C01786=1131.431,222.505,-66.418,-178.866,9.578,149.578
C01787=1131.435,222.257,-66.392,-178.868,9.575,149.578
C01788=1131.439,222.008,-66.366,-178.871,9.572,149.578
C01789=1131.445,221.760,-66.340,-178.874,9.569,149.578
C01790=1131.449,221.512,-66.313,-178.877,9.565,149.578
C01791=1131.453,221.263,-66.288,-178.880,9.562,149.578
C01792=1131.458,221.014,-66.261,-178.882,9.559,149.578
C01793=1131.462,220.765,-66.235,-178.885,9.556,149.578
C01794=1131.466,220.517,-66.209,-178.887,9.553,149.578
C01795=1131.471,220.269,-66.184,-178.890,9.550,149.578
C01796=1131.476,220.019,-66.157,-178.892,9.547,149.578
C01797=1131.480,219.771,-66.132,-178.895,9.544,149.577
C01798=1131.484,219.522,-66.105,-178.897,9.540,149.577
C01799=1131.488,219.274,-66.079,-178.899,9.537,149.577
C01800=1131.493,219.026,-66.054,-178.902,9.534,149.577
C01801=1131.498,218.776,-66.028,-178.904,9.531,149.577
C01802=1131.502,218.528,-66.002,-178.907,9.528,149.577
C01803=1131.506,218.279,-65.976,-178.910,9.525,149.577
C01804=1131.510,218.031,-65.950,-178.911,9.522,149.577
C01805=1131.515,217.783,-65.924,-178.914,9.519,149.577
C01806=1131.519,217.534,-65.899,-178.916,9.516,149.577
C01807=1131.524,217.285,-65.872,-178.918,9.513,149.576
C01808=1131.529,217.036,-65.846,-178.920,9.510,149.576
C01809=1131.533,216.788,-65.821,-178.923,9.507,149.576
C01810=1131.538,216.539,-65.795,-178.924,9.504,149.576
C01811=1131.542,216.290,-65.770,-178.927,9.501,149.576
C01812=1131.546,216.041,-65.744,-178.928,9.499,149.576
C01813=1131.551,215.793,-65.718,-178.931,9.495,149.576
C01814=1131.555,215.544,-65.693,-178.932,9.493,149.576
C01815=1131.559,215.296,-65.667,-178.934,9.490,149.575
C01816=1131.564,215.047,-65.642,-178.936,9.487,149.575
C01817=1131.569,214.798,-65.615,-178.938,9.484,149.575
C01818=1131.573,214.550,-65.589,-178.940,9.482,149.575
C01819=1131.578,214.301,-65.564,-178.942,9.479,149.575
C01820=1131.582,214.053,-65.538,-178.944,9.476,149.575
C01821=1131.587,213.804,-65.513,-178.945,9.474,149.574
C01822=1131.591,213.555,-65.487,-178.947,9.471,149.574
C01823=1131.596,213.307,-65.461,-178.949,9.469,149.574
C01824=1131.599,213.092,-65.440,-178.950,9.467,149.574
C01825=1131.603,212.878,-65.418,-178.951,9.464,149.574
C01826=1131.607,212.664,-65.395,-178.952,9.462,149.574
C01827=1131.611,212.450,-65.374,-178.954,9.460,149.574
C01828=1131.614,212.235,-65.351,-178.955,9.458,149.573
C01829=1131.618,212.021,-65.329,-178.957,9.456,149.573
C01830=1131.622,211.807,-65.307,-178.958,9.454,149.573
C01831=1131.626,211.592,-65.285,-178.960,9.452,149.573
C01832=1131.631,211.344,-65.259,-178.961,9.449,149.573
C01833=1131.634,211.096,-65.234,-178.963,9.446,149.573
C01834=1131.640,210.847,-65.210,-178.965,9.444,149.573
C01835=1131.644,210.598,-65.184,-178.967,9.442,149.573
C01836=1131.648,210.349,-65.158,-178.969,9.439,149.573
C01837=1131.653,210.101,-65.133,-178.970,9.437,149.572
C01838=1131.657,209.852,-65.107,-178.972,9.434,149.572
C01839=1131.662,209.603,-65.082,-178.975,9.431,149.572
C01840=1131.666,209.355,-65.057,-178.976,9.429,149.572
C01841=1131.671,209.106,-65.031,-178.979,9.427,149.572
C01842=1131.675,208.857,-65.005,-178.981,9.424,149.572
C01843=1131.680,208.608,-64.980,-178.983,9.422,149.572
C01844=1131.684,208.360,-64.955,-178.985,9.419,149.572
C01845=1131.689,208.112,-64.929,-178.988,9.416,149.572
C01846=1131.694,207.862,-64.904,-178.990,9.414,149.572
C01847=1131.697,207.614,-64.879,-178.992,9.411,149.572
C01848=1131.702,207.366,-64.854,-178.995,9.408,149.572
C01849=1131.706,207.116,-64.829,-178.997,9.406,149.572
C01850=1131.711,206.868,-64.803,-179.000,9.403,149.572
C01851=1131.715,206.619,-64.778,-179.003,9.400,149.572
C01852=1131.721,206.371,-64.753,-179.005,9.397,149.572
C01853=1131.725,206.122,-64.727,-179.008,9.395,149.573
C01854=1131.729,205.874,-64.702,-179.011,9.392,149.573
C01855=1131.733,205.624,-64.677,-179.013,9.389,149.573
C01856=1131.738,205.376,-64.652,-179.016,9.387,149.573
C01857=1131.743,205.127,-64.627,-179.019,9.384,149.573
C01858=1131.747,204.878,-64.601,-179.022,9.381,149.573
C01859=1131.751,204.630,-64.577,-179.024,9.378,149.573
C01860=1131.756,204.381,-64.551,-179.027,9.375,149.573
C01861=1131.761,204.132,-64.527,-179.031,9.372,149.573
C01862=1131.765,203.883,-64.501,-179.034,9.369,149.573
C01863=1131.770,203.635,-64.476,-179.036,9.366,149.573
C01864=1131.774,203.386,-64.451,-179.039,9.363,149.574
C01865=1131.779,203.137,-64.426,-179.043,9.360,149.574
C01866=1131.783,202.889,-64.401,-179.046,9.357,149.574
C01867=1131.787,202.640,-64.377,-179.050,9.353,149.574
C01868=1131.792,202.391,-64.351,-179.053,9.351,149.574
C01869=1131.797,202.143,-64.326,-179.056,9.347,149.574
C01870=1131.801,201.894,-64.302,-179.059,9.344,149.574
C01871=1131.805,201.646,-64.276,-179.063,9.341,149.575
C01872=1131.810,201.397,-64.252,-179.066,9.337,149.575
C01873=1131.814,201.148,-64.227,-179.070,9.334,149.575
C01874=1131.819,200.900,-64.202,-179.073,9.331,149.575
C01875=1131.823,200.650,-64.177,-179.077,9.328,149.575
C01876=1131.828,200.402,-64.153,-179.080,9.324,149.575
C01877=1131.833,200.152,-64.128,-179.084,9.321,149.576
C01878=1131.837,199.905,-64.103,-179.088,9.317,149.576
C01879=1131.842,199.656,-64.078,-179.091,9.314,149.576
C01880=1131.845,199.440,-64.057,-179.095,9.310,149.576
C01881=1131.849,199.227,-64.036,-179.098,9.308,149.576
C01882=1131.853,199.012,-64.015,-179.101,9.304,149.576
C01883=1131.857,198.798,-63.993,-179.104,9.301,149.576
C01884=1131.861,198.583,-63.972,-179.108,9.298,149.577
C01885=1131.864,198.369,-63.950,-179.111,9.295,149.577
C01886=1131.868,198.155,-63.930,-179.114,9.292,149.577
C01887=1131.872,197.941,-63.908,-179.118,9.288,149.577
C01888=1131.877,197.692,-63.884,-179.122,9.285,149.577
C01889=1131.882,197.443,-63.860,-179.126,9.281,149.578
C01890=1131.886,197.194,-63.834,-179.130,9.277,149.578
C01891=1131.890,196.946,-63.810,-179.134,9.273,149.578
C01892=1131.896,196.697,-63.786,-179.138,9.269,149.578
C01893=1131.899,196.448,-63.761,-179.142,9.265,149.578
C01894=1131.904,196.199,-63.737,-179.146,9.261,149.578
C01895=1131.909,195.951,-63.713,-179.147,9.259,149.578
C01896=1131.913,195.702,-63.688,-179.148,9.256,149.578
C01897=1131.918,195.453,-63.663,-179.150,9.254,149.578
C01898=1131.923,195.204,-63.640,-179.152,9.251,149.577
C01899=1131.927,194.955,-63.616,-179.153,9.248,149.577
C01900=1131.931,194.706,-63.591,-179.155,9.246,149.577
C01901=1131.936,194.458,-63.567,-179.156,9.244,149.577
C01902=1131.940,194.209,-63.543,-179.157,9.241,149.577
C01903=1131.945,193.960,-63.518,-179.159,9.239,149.577
C01904=1131.949,193.711,-63.494,-179.161,9.236,149.576
C01905=1131.954,193.463,-63.470,-179.163,9.234,149.576
C01906=1131.959,193.213,-63.446,-179.164,9.231,149.576
C01907=1131.963,192.965,-63.422,-179.166,9.229,149.576
C01908=1131.967,192.716,-63.397,-179.167,9.226,149.576
C01909=1131.972,192.467,-63.372,-179.169,9.224,149.576
C01910=1131.977,192.219,-63.348,-179.171,9.221,149.576
C01911=1131.981,191.970,-63.324,-179.173,9.218,149.576
C01912=1131.986,191.720,-63.300,-179.175,9.216,149.576
C01913=1131.990,191.472,-63.276,-179.177,9.213,149.575
C01914=1131.995,191.224,-63.252,-179.179,9.211,149.575
C01915=1131.999,190.975,-63.228,-179.181,9.208,149.575
C01916=1132.005,190.726,-63.204,-179.183,9.205,149.575
C01917=1132.008,190.477,-63.179,-179.184,9.203,149.575
C01918=1132.013,190.228,-63.155,-179.187,9.200,149.575
C01919=1132.018,189.980,-63.131,-179.189,9.197,149.575
C01920=1132.023,189.731,-63.107,-179.191,9.195,149.575
C01921=1132.027,189.482,-63.083,-179.193,9.192,149.575
C01922=1132.031,189.234,-63.059,-179.195,9.189,149.575
C01923=1132.035,188.984,-63.035,-179.198,9.186,149.575
C01924=1132.041,188.735,-63.011,-179.200,9.184,149.575
C01925=1132.045,188.487,-62.987,-179.202,9.181,149.575
C01926=1132.050,188.238,-62.963,-179.205,9.178,149.575
C01927=1132.054,187.989,-62.939,-179.207,9.176,149.575
C01928=1132.058,187.741,-62.915,-179.209,9.172,149.575
C01929=1132.063,187.491,-62.891,-179.212,9.169,149.575
C01930=1132.068,187.243,-62.867,-179.213,9.167,149.574
C01931=1132.072,186.993,-62.843,-179.216,9.164,149.574
C01932=1132.077,186.745,-62.819,-179.219,9.161,149.574
C01933=1132.081,186.496,-62.796,-179.221,9.158,149.574
C01934=1132.086,186.248,-62.772,-179.224,9.155,149.574
C01935=1132.090,185.999,-62.748,-179.226,9.153,149.574
C01936=1132.095,185.784,-62.728,-179.228,9.149,149.574
C01937=1132.098,185.569,-62.707,-179.230,9.147,149.574
C01938=1132.102,185.355,-62.686,-179.233,9.144,149.574
C01939=1132.106,185.140,-62.666,-179.235,9.142,149.574
C01940=1132.111,184.926,-62.645,-179.237,9.140,149.574
C01941=1132.114,184.712,-62.625,-179.240,9.137,149.574
C01942=1132.118,184.498,-62.604,-179.241,9.134,149.574
C01943=1132.122,184.282,-62.584,-179.244,9.131,149.574
C01944=1132.126,184.034,-62.560,-179.247,9.128,149.574
C01945=1132.131,183.785,-62.537,-179.249,9.125,149.575
C01946=1132.136,183.536,-62.513,-179.253,9.121,149.574
C01947=1132.140,183.287,-62.489,-179.255,9.118,149.574
C01948=1132.145,183.038,-62.466,-179.258,9.116,149.575
C01949=1132.149,182.790,-62.442,-179.261,9.113,149.575
C01950=1132.154,182.541,-62.418,-179.264,9.109,149.574
C01951=1132.159,182.292,-62.395,-179.267,9.106,149.575
C01952=1132.163,182.043,-62.371,-179.269,9.103,149.575
C01953=1132.168,181.794,-62.348,-179.272,9.099,149.575
C01954=1132.173,181.545,-62.324,-179.275,9.096,149.575
C01955=1132.177,181.297,-62.300,-179.279,9.092,149.575
C01956=1132.182,181.048,-62.277,-179.282,9.090,149.575
C01957=1132.186,180.799,-62.254,-179.285,9.086,149.575
C01958=1132.191,180.550,-62.230,-179.288,9.082,149.575
C01959=1132.195,180.302,-62.206,-179.291,9.079,149.575
C01960=1132.199,180.053,-62.183,-179.294,9.075,149.575
C01961=1132.204,179.804,-62.160,-179.298,9.072,149.575
C01962=1132.209,179.555,-62.137,-179.300,9.069,149.575
C01963=1132.214,179.306,-62.113,-179.304,9.065,149.575
C01964=1132.218,179.057,-62.090,-179.306,9.062,149.575
C01965=1132.223,178.808,-62.067,-179.308,9.058,149.575
C01966=1132.227,178.559,-62.042,-179.311,9.055,149.575
C01967=1132.231,178.310,-62.020,-179.312,9.053,149.575
C01968=1132.236,178.061,-61.996,-179.315,9.050,149.575
C01969=1132.241,177.812,-61.973,-179.317,9.047,149.575
C01970=1132.245,177.563,-61.950,-179.319,9.044,149.574
C01971=1132.250,177.314,-61.926,-179.321,9.041,149.574
C01972=1132.254,177.066,-61.903,-179.323,9.038,149.574
C01973=1132.259,176.817,-61.880,-179.325,9.035,149.574
C01974=1132.264,176.568,-61.857,-179.327,9.033,149.574
C01975=1132.269,176.319,-61.834,-179.330,9.029,149.574
C01976=1132.273,176.071,-61.811,-179.332,9.026,149.574
C01977=1132.277,175.821,-61.788,-179.334,9.024,149.574
C01978=1132.282,175.572,-61.764,-179.336,9.020,149.574
C01979=1132.287,175.323,-61.741,-179.338,9.017,149.573
C01980=1132.291,175.075,-61.718,-179.340,9.015,149.573
C01981=1132.296,174.826,-61.695,-179.343,9.012,149.573
C01982=1132.301,174.577,-61.672,-179.345,9.008,149.573
C01983=1132.305,174.328,-61.648,-179.347,9.005,149.573
C01984=1132.310,174.079,-61.626,-179.349,9.003,149.573
C01985=1132.314,173.830,-61.603,-179.352,9.000,149.573
C01986=1132.319,173.581,-61.580,-179.354,8.996,149.573
C01987=1132.323,173.332,-61.557,-179.356,8.994,149.573
C01988=1132.328,173.084,-61.534,-179.358,8.991,149.573
C01989=1132.333,172.835,-61.511,-179.361,8.988,149.573
C01990=1132.337,172.586,-61.488,-179.363,8.984,149.572
C01991=1132.342,172.336,-61.465,-179.365,8.981,149.572
C01992=1132.346,172.123,-61.445,-179.367,8.979,149.572
C01993=1132.350,171.908,-61.425,-179.369,8.976,149.572
C01994=1132.354,171.693,-61.406,-179.371,8.974,149.572
C01995=1132.358,171.478,-61.386,-179.373,8.970,149.572
C01996=1132.362,171.264,-61.366,-179.375,8.968,149.572
C01997=1132.366,171.049,-61.346,-179.377,8.966,149.572
C01998=1132.370,170.835,-61.327,-179.380,8.963,149.572
C01999=1132.373,170.620,-61.307,-179.381,8.960,149.572
C02000=1132.379,170.371,-61.284,-179.383,8.957,149.572
C02001=1132.383,170.122,-61.261,-179.386,8.954,149.572
C02002=1132.388,169.873,-61.239,-179.388,8.951,149.572
C02003=1132.392,169.624,-61.216,-179.390,8.948,149.572
C02004=1132.397,169.376,-61.193,-179.393,8.945,149.571
C02005=1132.402,169.126,-61.171,-179.395,8.942,149.571
C02006=1132.406,168.878,-61.148,-179.398,8.939,149.571
C02007=1132.411,168.629,-61.125,-179.400,8.936,149.571
C02008=1132.415,168.380,-61.103,-179.402,8.932,149.571
C02009=1132.420,168.131,-61.079,-179.405,8.929,149.571
C02010=1132.424,167.882,-61.057,-179.407,8.926,149.571
C02011=1132.430,167.633,-61.034,-179.410,8.923,149.571
C02012=1132.434,167.384,-61.012,-179.412,8.920,149.571
C02013=1132.439,167.135,-60.989,-179.414,8.916,149.571
C02014=1132.443,166.887,-60.967,-179.417,8.913,149.571
C02015=1132.448,166.637,-60.944,-179.419,8.910,149.571
C02016=1132.452,166.388,-60.921,-179.422,8.907,149.571
C02017=1132.458,166.139,-60.899,-179.424,8.903,149.570
C02018=1132.462,165.891,-60.876,-179.427,8.900,149.570
C02019=1132.466,165.641,-60.854,-179.429,8.897,149.570
C02020=1132.471,165.393,-60.831,-179.432,8.894,149.570
C02021=1132.476,165.144,-60.809,-179.434,8.891,149.570
C02022=1132.481,164.894,-60.786,-179.436,8.887,149.570
C02023=1132.485,164.646,-60.764,-179.439,8.884,149.570
C02024=1132.489,164.397,-60.742,-179.441,8.881,149.570
C02025=1132.494,164.148,-60.719,-179.444,8.878,149.570
C02026=1132.499,163.899,-60.697,-179.446,8.875,149.570
C02027=1132.503,163.650,-60.675,-179.448,8.872,149.570
C02028=1132.508,163.401,-60.652,-179.451,8.868,149.570
C02029=1132.513,163.152,-60.630,-179.453,8.865,149.570
C02030=1132.517,162.903,-60.607,-179.457,8.861,149.569
C02031=1132.522,162.654,-60.585,-179.459,8.858,149.569
C02032=1132.527,162.405,-60.563,-179.461,8.855,149.569
C02033=1132.531,162.156,-60.541,-179.464,8.852,149.569
C02034=1132.536,161.907,-60.518,-179.466,8.849,149.569
C02035=1132.540,161.658,-60.496,-179.468,8.845,149.569
C02036=1132.545,161.409,-60.474,-179.472,8.841,149.569
C02037=1132.550,161.160,-60.452,-179.474,8.838,149.569
C02038=1132.555,160.912,-60.429,-179.477,8.835,149.569
C02039=1132.559,160.662,-60.407,-179.479,8.832,149.569
C02040=1132.563,160.413,-60.385,-179.482,8.828,149.569
C02041=1132.568,160.164,-60.363,-179.484,8.825,149.569
C02042=1132.573,159.915,-60.341,-179.487,8.821,149.568
C02043=1132.578,159.667,-60.318,-179.489,8.818,149.568
C02044=1132.582,159.417,-60.296,-179.492,8.814,149.568
C02045=1132.587,159.169,-60.274,-179.495,8.811,149.568
C02046=1132.591,158.919,-60.252,-179.497,8.808,149.568
C02047=1132.596,158.671,-60.231,-179.500,8.804,149.568
C02048=1132.604,158.252,-60.193,-179.504,8.798,149.568
C02049=1132.612,157.833,-60.156,-179.508,8.792,149.568
C02050=1132.620,157.416,-60.119,-179.513,8.786,149.568
C02051=1132.628,156.997,-60.082,-179.517,8.780,149.567
C02052=1132.632,156.748,-60.061,-179.520,8.777,149.567
C02053=1132.637,156.499,-60.039,-179.523,8.773,149.567
C02054=1132.642,156.250,-60.017,-179.525,8.770,149.567
C02055=1132.646,156.001,-59.995,-179.528,8.766,149.567
C02056=1132.651,155.752,-59.973,-179.531,8.763,149.567
C02057=1132.655,155.503,-59.951,-179.534,8.759,149.567
C02058=1132.660,155.254,-59.930,-179.536,8.755,149.567
C02059=1132.665,155.006,-59.908,-179.538,8.752,149.567
C02060=1132.669,154.756,-59.887,-179.542,8.748,149.567
C02061=1132.674,154.507,-59.865,-179.544,8.744,149.566
C02062=1132.678,154.258,-59.843,-179.547,8.741,149.566
C02063=1132.683,154.009,-59.821,-179.550,8.737,149.566
C02064=1132.688,153.760,-59.799,-179.552,8.734,149.566
C02065=1132.692,153.511,-59.777,-179.555,8.730,149.566
C02066=1132.698,153.262,-59.756,-179.557,8.726,149.566
C02067=1132.703,153.013,-59.735,-179.560,8.722,149.566
C02068=1132.707,152.764,-59.713,-179.563,8.719,149.566
C02069=1132.712,152.515,-59.691,-179.566,8.715,149.566
C02070=1132.717,152.266,-59.670,-179.569,8.711,149.566
C02071=1132.721,152.016,-59.648,-179.571,8.708,149.565
C02072=1132.726,151.768,-59.626,-179.574,8.704,149.565
C02073=1132.731,151.519,-59.605,-179.577,8.700,149.565
C02074=1132.735,151.269,-59.583,-179.579,8.696,149.565
C02075=1132.740,151.021,-59.562,-179.582,8.693,149.565
C02076=1132.745,150.772,-59.541,-179.585,8.688,149.565
C02077=1132.749,150.522,-59.519,-179.588,8.685,149.565
C02078=1132.754,150.274,-59.497,-179.590,8.681,149.565
C02079=1132.759,150.024,-59.477,-179.594,8.677,149.564
C02080=1132.782,148.793,-59.374,-178.796,7.149,148.985
C02081=1132.787,148.545,-59.352,-178.799,7.147,148.985
C02082=1132.792,148.296,-59.332,-178.802,7.145,148.985
C02083=1132.796,148.046,-59.310,-178.805,7.143,148.986
C02084=1132.801,147.797,-59.289,-178.807,7.141,148.986
C02085=1132.805,147.548,-59.268,-178.811,7.139,148.986
C02086=1132.811,147.299,-59.247,-178.813,7.137,148.987
C02087=1132.816,147.050,-59.226,-178.816,7.135,148.987
C02088=1132.820,146.801,-59.205,-178.819,7.132,148.987
C02089=1132.825,146.552,-59.184,-178.822,7.131,148.988
C02090=1132.830,146.303,-59.164,-178.824,7.129,148.988
C02091=1132.834,146.053,-59.143,-178.828,7.127,148.988
C02092=1132.839,145.805,-59.121,-178.830,7.125,148.989
C02093=1132.843,145.556,-59.100,-178.833,7.123,148.989
C02094=1132.849,145.306,-59.080,-178.836,7.120,148.989
C02095=1132.853,145.057,-59.059,-178.839,7.119,148.990
C02096=1132.858,144.808,-59.038,-178.841,7.117,148.990
C02097=1132.863,144.559,-59.018,-178.845,7.114,148.991
C02098=1132.867,144.311,-58.996,-178.847,7.113,148.991
C02099=1132.872,144.062,-58.976,-178.850,7.111,148.991
C02100=1132.877,143.812,-58.955,-178.853,7.108,148.991
C02101=1132.882,143.563,-58.934,-178.856,7.106,148.992
C02102=1132.886,143.313,-58.913,-178.858,7.105,148.992
C02103=1132.891,143.065,-58.893,-178.862,7.102,148.993
C02104=1132.896,142.815,-58.872,-178.864,7.101,148.993
C02105=1132.900,142.566,-58.851,-178.867,7.098,148.993
C02106=1132.905,142.317,-58.830,-178.869,7.097,148.994
C02107=1132.910,142.068,-58.810,-178.873,7.094,148.994
C02108=1132.915,141.819,-58.789,-178.875,7.093,148.994
C02109=1132.919,141.570,-58.769,-178.878,7.091,148.995
C02110=1132.924,141.321,-58.748,-178.881,7.088,148.995
C02111=1132.929,141.072,-58.727,-178.884,7.087,148.995
C02112=1132.933,140.823,-58.707,-178.886,7.085,148.996
C02113=1132.939,140.573,-58.686,-178.889,7.083,148.996
C02114=1132.943,140.325,-58.666,-178.892,7.080,148.996
C02115=1132.947,140.076,-58.645,-178.895,7.079,148.997
C02116=1132.953,139.826,-58.624,-178.898,7.077,148.997
C02117=1132.957,139.577,-58.604,-178.901,7.075,148.998
C02118=1132.962,139.328,-58.584,-178.904,7.073,148.998
C02119=1132.967,139.079,-58.563,-178.907,7.071,148.998
C02120=1132.971,138.830,-58.543,-178.909,7.069,148.999
C02121=1132.976,138.581,-58.523,-178.912,7.067,148.999
C02122=1132.981,138.331,-58.502,-178.915,7.065,148.999
C02123=1132.985,138.082,-58.481,-178.918,7.063,149.000
C02124=1132.990,137.833,-58.461,-178.920,7.062,149.000
C02125=1132.995,137.584,-58.440,-178.924,7.059,149.000
C02126=1133.000,137.335,-58.420,-178.926,7.057,149.001
C02127=1133.004,137.086,-58.400,-178.929,7.056,149.001
C02128=1133.010,136.837,-58.379,-178.931,7.054,149.001
C02129=1133.014,136.588,-58.359,-178.935,7.051,149.002
C02130=1133.019,136.339,-58.339,-178.937,7.049,149.002
C02131=1133.024,136.090,-58.319,-178.940,7.048,149.003
C02132=1133.029,135.840,-58.298,-178.943,7.046,149.003
C02133=1133.033,135.591,-58.278,-178.946,7.044,149.003
C02134=1133.038,135.342,-58.258,-178.949,7.042,149.004
C02135=1133.042,135.093,-58.237,-178.952,7.040,149.004
C02136=1133.048,134.844,-58.217,-178.954,7.038,149.005
C02137=1133.052,134.594,-58.197,-178.958,7.036,149.005
C02138=1133.057,134.346,-58.177,-178.960,7.034,149.005
C02139=1133.062,134.097,-58.156,-178.963,7.032,149.005
C02140=1133.067,133.847,-58.137,-178.965,7.031,149.006
C02141=1133.072,133.598,-58.116,-178.969,7.028,149.006
C02142=1133.076,133.349,-58.096,-178.971,7.026,149.007
C02143=1133.081,133.100,-58.076,-178.974,7.025,149.007
C02144=1133.085,132.851,-58.055,-178.977,7.023,149.007
C02145=1133.091,132.602,-58.036,-178.980,7.021,149.008
C02146=1133.095,132.353,-58.016,-178.983,7.019,149.008
C02147=1133.100,132.103,-57.996,-178.986,7.017,149.009
C02148=1133.105,131.854,-57.975,-178.988,7.015,149.009
C02149=1133.110,131.585,-57.954,-178.991,7.014,149.009
C02150=1133.115,131.317,-57.932,-178.994,7.011,149.010
C02151=1133.120,131.048,-57.911,-178.997,7.010,149.010
C02152=1133.125,130.780,-57.890,-179.000,7.007,149.011
C02153=1133.130,130.531,-57.869,-179.003,7.005,149.011
C02154=1133.136,130.282,-57.849,-179.006,7.004,149.011
C02155=1133.140,130.033,-57.829,-179.009,7.002,149.012
C02156=1133.145,129.783,-57.809,-179.012,6.999,149.012
C02157=1133.149,129.534,-57.789,-179.014,6.997,149.012
C02158=1133.155,129.285,-57.770,-179.017,6.996,149.013
C02159=1133.159,129.036,-57.750,-179.020,6.994,149.013
C02160=1133.164,128.787,-57.730,-179.022,6.992,149.014
C02161=1133.169,128.537,-57.710,-179.026,6.990,149.014
C02162=1133.174,128.289,-57.690,-179.028,6.988,149.014
C02163=1133.178,128.039,-57.670,-179.031,6.987,149.015
C02164=1133.183,127.790,-57.651,-179.034,6.985,149.015
C02165=1133.188,127.541,-57.630,-179.037,6.983,149.016
C02166=1133.193,127.292,-57.611,-179.039,6.981,149.016
C02167=1133.198,127.042,-57.591,-179.043,6.979,149.016
C02168=1133.202,126.793,-57.571,-179.045,6.977,149.017
C02169=1133.207,126.544,-57.551,-179.048,6.976,149.017
C02170=1133.212,126.295,-57.532,-179.051,6.974,149.018
C02171=1133.217,126.045,-57.512,-179.054,6.972,149.018
C02172=1133.221,125.796,-57.492,-179.056,6.971,149.018
C02173=1133.226,125.548,-57.473,-179.060,6.968,149.019
C02174=1133.231,125.298,-57.454,-179.062,6.966,149.019
C02175=1133.235,125.049,-57.434,-179.065,6.965,149.019
C02176=1133.240,124.800,-57.414,-179.068,6.963,149.020
C02177=1133.245,124.551,-57.394,-179.071,6.961,149.020
C02178=1133.250,124.301,-57.375,-179.073,6.960,149.021
C02179=1133.255,124.052,-57.355,-179.076,6.957,149.021
C02180=1133.260,123.803,-57.336,-179.079,6.955,149.021
C02181=1133.264,123.554,-57.315,-179.082,6.953,149.022
C02182=1133.268,123.305,-57.296,-179.084,6.952,149.022
C02183=1133.274,123.056,-57.277,-179.087,6.950,149.022
C02184=1133.279,122.806,-57.257,-179.090,6.948,149.023
C02185=1133.283,122.557,-57.238,-179.092,6.947,149.023
C02186=1133.289,122.308,-57.218,-179.096,6.944,149.024
C02187=1133.293,122.058,-57.199,-179.099,6.943,149.024
C02188=1133.298,121.810,-57.180,-179.101,6.941,149.024
C02189=1133.303,121.560,-57.160,-179.104,6.939,149.025
C02190=1133.307,121.311,-57.140,-179.107,6.937,149.025
C02191=1133.313,121.062,-57.121,-179.109,6.936,149.026
C02192=1133.317,120.813,-57.101,-179.112,6.934,149.026
C02193=1133.322,120.564,-57.082,-179.115,6.932,149.026
C02194=1133.327,120.315,-57.063,-179.118,6.930,149.027
C02195=1133.331,120.065,-57.043,-179.121,6.928,149.027
C02196=1133.337,119.816,-57.024,-179.124,6.927,149.028
C02197=1133.341,119.567,-57.005,-179.126,6.925,149.028
C02198=1133.346,119.318,-56.985,-179.129,6.923,149.029
C02199=1133.351,119.069,-56.966,-179.132,6.922,149.029
C02200=1133.356,118.819,-56.948,-179.135,6.920,149.029
C02201=1133.360,118.570,-56.928,-179.137,6.918,149.030
C02202=1133.365,118.320,-56.908,-179.140,6.916,149.030
C02203=1133.371,118.071,-56.889,-179.143,6.914,149.031
C02204=1133.375,117.822,-56.870,-179.146,6.912,149.031
C02205=1133.380,117.573,-56.851,-179.149,6.911,149.031
C02206=1133.385,117.324,-56.831,-179.152,6.909,149.032
C02207=1133.389,117.075,-56.812,-179.154,6.907,149.032
C02208=1133.394,116.826,-56.793,-179.157,6.906,149.033
C02209=1133.400,116.576,-56.774,-179.160,6.904,149.033
C02210=1133.404,116.327,-56.755,-179.163,6.902,149.033
C02211=1133.409,116.078,-56.736,-179.165,6.901,149.034
C02212=1133.413,115.829,-56.717,-179.168,6.899,149.034
C02213=1133.418,115.580,-56.697,-179.171,6.897,149.035
C02214=1133.423,115.330,-56.679,-179.174,6.895,149.035
C02215=1133.428,115.081,-56.660,-179.177,6.893,149.035
C02216=1133.433,114.832,-56.640,-179.180,6.891,149.036
C02217=1133.438,114.583,-56.621,-179.183,6.890,149.036
C02218=1133.442,114.333,-56.603,-179.185,6.888,149.037
C02219=1133.448,114.084,-56.583,-179.188,6.887,149.037
C02220=1133.452,113.835,-56.564,-179.191,6.885,149.038
C02221=1133.457,113.586,-56.545,-179.194,6.883,149.038
C02222=1133.462,113.337,-56.527,-179.196,6.882,149.038
C02223=1133.467,113.087,-56.507,-179.199,6.880,149.039
C02224=1133.471,112.838,-56.489,-179.202,6.878,149.039
C02225=1133.476,112.588,-56.470,-179.205,6.877,149.040
C02226=1133.482,112.339,-56.450,-179.207,6.875,149.040
C02227=1133.486,112.090,-56.431,-179.210,6.873,149.040
C02228=1133.491,111.841,-56.413,-179.213,6.872,149.041
C02229=1133.496,111.592,-56.394,-179.216,6.870,149.041
C02230=1133.501,111.342,-56.375,-179.219,6.867,149.042
C02231=1133.506,111.093,-56.356,-179.222,6.866,149.042
C02232=1133.510,110.844,-56.337,-179.224,6.864,149.043
C02233=1133.515,110.595,-56.319,-179.227,6.862,149.043
C02234=1133.520,110.346,-56.300,-179.230,6.861,149.043
C02235=1133.525,110.096,-56.281,-179.233,6.859,149.044
C02236=1133.530,109.847,-56.262,-179.235,6.857,149.044
C02237=1133.535,109.597,-56.243,-179.238,6.856,149.045
C02238=1133.539,109.349,-56.225,-179.241,6.854,149.045
C02239=1133.545,109.099,-56.206,-179.243,6.852,149.045
C02240=1133.549,108.850,-56.187,-179.247,6.851,149.046
C02241=1133.554,108.601,-56.169,-179.249,6.849,149.046
C02242=1133.559,108.352,-56.150,-179.252,6.848,149.047
C02243=1133.563,108.102,-56.132,-179.255,6.846,149.047
C02244=1133.569,107.853,-56.112,-179.258,6.844,149.048
C02245=1133.574,107.604,-56.094,-179.260,6.843,149.048
C02246=1133.578,107.355,-56.075,-179.263,6.841,149.048
C02247=1133.583,107.105,-56.057,-179.266,6.839,149.049
C02248=1133.588,106.856,-56.039,-179.269,6.838,149.049
C02249=1133.592,106.607,-56.020,-179.271,6.836,149.050
C02250=1133.598,106.357,-56.001,-179.274,6.834,149.050
C02251=1133.603,106.108,-55.983,-179.277,6.833,149.051
C02252=1133.607,105.859,-55.964,-179.279,6.831,149.051
C02253=1133.613,105.590,-55.944,-179.283,6.830,149.052
C02254=1133.618,105.322,-55.925,-179.286,6.827,149.052
C02255=1133.623,105.054,-55.904,-179.289,6.826,149.052
C02256=1133.628,104.786,-55.884,-179.292,6.824,149.053
C02257=1133.633,104.536,-55.866,-179.294,6.822,149.053
C02258=1133.638,104.286,-55.847,-179.297,6.821,149.054
C02259=1133.643,104.038,-55.829,-179.300,6.819,149.054
C02260=1133.647,103.788,-55.810,-179.303,6.818,149.055
C02261=1133.652,103.539,-55.792,-179.306,6.816,149.055
C02262=1133.658,103.289,-55.774,-179.308,6.814,149.056
C02263=1133.662,103.041,-55.755,-179.311,6.813,149.056
C02264=1133.667,102.791,-55.737,-179.314,6.811,149.056
C02265=1133.672,102.542,-55.719,-179.317,6.809,149.057
C02266=1133.677,102.292,-55.700,-179.319,6.808,149.057
C02267=1133.682,102.044,-55.682,-179.322,6.806,149.058
C02268=1133.687,101.794,-55.664,-179.325,6.804,149.058
C02269=1133.691,101.545,-55.645,-179.328,6.803,149.059
C02270=1133.696,101.295,-55.627,-179.331,6.801,149.059
C02271=1133.702,101.046,-55.609,-179.334,6.800,149.059
C02272=1133.707,100.797,-55.591,-179.336,6.798,149.060
C02273=1133.711,100.548,-55.573,-179.339,6.796,149.060
C02274=1133.715,100.298,-55.554,-179.342,6.795,149.061
C02275=1133.720,100.049,-55.536,-179.344,6.793,149.061
C02276=1133.725,99.800,-55.518,-179.347,6.792,149.062
C02277=1133.730,99.551,-55.500,-179.349,6.790,149.062
C02278=1133.736,99.301,-55.481,-179.352,6.789,149.062
C02279=1133.740,99.051,-55.463,-179.355,6.787,149.063
C02280=1133.745,98.802,-55.445,-179.358,6.786,149.063
C02281=1133.750,98.553,-55.427,-179.361,6.784,149.064
C02282=1133.755,98.304,-55.409,-179.364,6.782,149.064
C02283=1133.760,98.055,-55.391,-179.366,6.781,149.065
C02284=1133.765,97.806,-55.373,-179.369,6.779,149.065
C02285=1133.770,97.556,-55.355,-179.372,6.777,149.066
C02286=1133.774,97.307,-55.337,-179.374,6.776,149.066
C02287=1133.779,97.057,-55.319,-179.377,6.774,149.066
C02288=1133.784,96.808,-55.301,-179.380,6.773,149.067
C02289=1133.789,96.559,-55.283,-179.383,6.771,149.067
C02290=1133.794,96.310,-55.265,-179.386,6.769,149.068
C02291=1133.799,96.061,-55.247,-179.389,6.768,149.068
C02292=1133.803,95.811,-55.229,-179.391,6.766,149.069
C02293=1133.808,95.562,-55.211,-179.394,6.765,149.069
C02294=1133.813,95.313,-55.193,-179.396,6.764,149.070
C02295=1133.818,95.063,-55.175,-179.400,6.762,149.070
C02296=1133.823,94.813,-55.157,-179.402,6.761,149.071
C02297=1133.828,94.564,-55.139,-179.405,6.759,149.071
C02298=1133.833,94.315,-55.121,-179.408,6.757,149.071
C02299=1133.838,94.066,-55.103,-179.410,6.756,149.072
C02300=1133.842,93.817,-55.085,-179.413,6.754,149.072
C02301=1133.848,93.567,-55.068,-179.416,6.752,149.073
C02302=1133.853,93.318,-55.050,-179.419,6.751,149.073
C02303=1133.857,93.069,-55.032,-179.422,6.749,149.074
C02304=1133.862,92.819,-55.014,-179.424,6.748,149.074
C02305=1133.867,92.570,-54.996,-179.427,6.747,149.075
C02306=1133.873,92.320,-54.979,-179.430,6.745,149.075
C02307=1133.877,92.071,-54.961,-179.432,6.744,149.075
C02308=1133.882,91.822,-54.943,-179.435,6.742,149.076
C02309=1133.887,91.573,-54.925,-179.438,6.740,149.076
C02310=1133.892,91.323,-54.908,-179.441,6.739,149.077
C02311=1133.897,91.074,-54.890,-179.444,6.737,149.077
C02312=1133.902,90.825,-54.872,-179.446,6.736,149.078
C02313=1133.906,90.576,-54.854,-179.449,6.735,149.078
C02314=1133.912,90.326,-54.837,-179.451,6.733,149.079
C02315=1133.917,90.077,-54.819,-179.454,6.731,149.079
C02316=1133.922,89.828,-54.801,-179.457,6.730,149.080
C02317=1133.926,89.578,-54.784,-179.460,6.728,149.080
C02318=1133.931,89.329,-54.766,-179.463,6.727,149.081
C02319=1133.936,89.079,-54.749,-179.466,6.725,149.081
C02320=1133.941,88.830,-54.731,-179.468,6.723,149.081
C02321=1133.946,88.581,-54.713,-179.470,6.723,149.082
C02322=1133.951,88.331,-54.696,-179.473,6.721,149.082
C02323=1133.955,88.082,-54.678,-179.476,6.720,149.083
C02324=1133.961,87.832,-54.661,-179.479,6.718,149.083
C02325=1133.965,87.583,-54.643,-179.482,6.716,149.084
C02326=1133.970,87.334,-54.625,-179.485,6.715,149.084
C02327=1133.975,87.085,-54.609,-179.487,6.713,149.085
C02328=1133.980,86.835,-54.591,-179.490,6.711,149.085
C02329=1133.985,86.586,-54.573,-179.493,6.711,149.086
C02330=1133.990,86.337,-54.555,-179.496,6.709,149.086
C02331=1133.994,86.087,-54.539,-179.498,6.708,149.087
C02332=1133.999,85.838,-54.521,-179.501,6.706,149.087
C02333=1134.005,85.589,-54.504,-179.504,6.704,149.087
C02334=1134.010,85.340,-54.486,-179.506,6.703,149.088
C02335=1134.015,85.090,-54.469,-179.509,6.702,149.088
C02336=1134.019,84.841,-54.451,-179.512,6.700,149.089
C02337=1134.025,84.591,-54.434,-179.515,6.699,149.089
C02338=1134.029,84.342,-54.417,-179.517,6.697,149.090
C02339=1134.034,84.092,-54.399,-179.520,6.695,149.090
C02340=1134.039,83.843,-54.382,-179.523,6.694,149.091
C02341=1134.043,83.594,-54.365,-179.525,6.693,149.091
C02342=1134.049,83.345,-54.348,-179.528,6.692,149.092
C02343=1134.054,83.095,-54.330,-179.531,6.690,149.092
C02344=1134.059,82.846,-54.313,-179.534,6.688,149.092
C02345=1134.064,82.596,-54.296,-179.536,6.687,149.093
C02346=1134.068,82.347,-54.279,-179.540,6.685,149.094
C02347=1134.073,82.098,-54.261,-179.542,6.685,149.094
C02348=1134.078,81.848,-54.244,-179.545,6.683,149.094
C02349=1134.084,81.599,-54.228,-179.547,6.681,149.095
C02350=1134.088,81.350,-54.210,-179.550,6.680,149.095
C02351=1134.093,81.100,-54.193,-179.553,6.678,149.096
C02352=1134.098,80.851,-54.176,-179.555,6.677,149.096
C02353=1134.103,80.601,-54.158,-179.558,6.676,149.097
C02354=1134.108,80.353,-54.141,-179.561,6.674,149.097
C02355=1134.113,80.103,-54.124,-179.564,6.672,149.098
C02356=1134.118,79.853,-54.107,-179.567,6.671,149.098
C02357=1134.123,79.584,-54.089,-179.570,6.670,149.099
C02358=1134.129,79.316,-54.070,-179.572,6.668,149.099
C02359=1134.134,79.048,-54.052,-179.576,6.667,149.100
C02360=1134.140,78.780,-54.033,-179.578,6.665,149.100
C02361=1134.144,78.531,-54.017,-179.581,6.663,149.101
C02362=1134.149,78.281,-53.999,-179.583,6.662,149.101
C02363=1134.154,78.031,-53.983,-179.586,6.661,149.102
C02364=1134.160,77.782,-53.966,-179.589,6.660,149.102
C02365=1134.164,77.533,-53.949,-179.592,6.658,149.103
C02366=1134.169,77.283,-53.932,-179.594,6.657,149.103
C02367=1134.173,77.034,-53.914,-179.597,6.655,149.103
C02368=1134.179,76.785,-53.898,-179.600,6.654,149.104
C02369=1134.184,76.536,-53.881,-179.603,6.652,149.105
C02370=1134.189,76.286,-53.864,-179.606,6.651,149.105
C02371=1134.193,76.036,-53.847,-179.608,6.650,149.105
C02372=1134.198,75.788,-53.831,-179.611,6.648,149.106
C02373=1134.204,75.538,-53.813,-179.614,6.647,149.106
C02374=1134.208,75.288,-53.797,-179.616,6.645,149.107
C02375=1134.214,75.039,-53.780,-179.619,6.645,149.107
C02376=1134.218,74.790,-53.763,-179.621,6.643,149.108
C02377=1134.223,74.540,-53.747,-179.625,6.642,149.108
C02378=1134.228,74.290,-53.729,-179.627,6.640,149.109
C02379=1134.233,74.042,-53.713,-179.630,6.639,149.109
C02380=1134.238,73.792,-53.696,-179.632,6.637,149.110
C02381=1134.243,73.542,-53.679,-179.635,6.636,149.110
C02382=1134.248,73.294,-53.663,-179.638,6.635,149.111
C02383=1134.253,73.044,-53.645,-179.640,6.634,149.111
C02384=1134.258,72.794,-53.629,-179.643,6.632,149.112
C02385=1134.263,72.546,-53.612,-179.646,6.630,149.112
C02386=1134.268,72.296,-53.595,-179.649,6.629,149.113
C02387=1134.273,72.046,-53.579,-179.651,6.628,149.113
C02388=1134.278,71.797,-53.562,-179.654,6.627,149.114
C02389=1134.283,71.548,-53.545,-179.657,6.625,149.114
C02390=1134.288,71.298,-53.529,-179.660,6.623,149.115
C02391=1134.293,71.049,-53.513,-179.662,6.623,149.115
C02392=1134.297,70.799,-53.496,-179.665,6.621,149.116
C02393=1134.303,70.550,-53.479,-179.668,6.620,149.116
C02394=1134.307,70.301,-53.462,-179.670,6.618,149.116
C02395=1134.312,70.051,-53.446,-179.673,6.617,149.117
C02396=1134.318,69.802,-53.429,-179.676,6.616,149.118
C02397=1134.323,69.552,-53.413,-179.679,6.614,149.118
C02398=1134.328,69.303,-53.397,-179.681,6.613,149.118
C02399=1134.332,69.054,-53.380,-179.684,6.612,149.119
C02400=1134.337,68.804,-53.363,-179.687,6.610,149.120
C02401=1134.343,68.555,-53.347,-179.689,6.609,149.120
C02402=1134.347,68.305,-53.330,-179.692,6.608,149.120
C02403=1134.352,68.056,-53.314,-179.695,6.607,149.121
C02404=1134.357,67.807,-53.297,-179.698,6.605,149.121
C02405=1134.363,67.557,-53.281,-179.700,6.604,149.122
C02406=1134.367,67.308,-53.265,-179.702,6.602,149.122
C02407=1134.372,67.058,-53.248,-179.705,6.601,149.123
C02408=1134.377,66.809,-53.232,-179.708,6.600,149.123
C02409=1134.382,66.559,-53.216,-179.711,6.599,149.124
C02410=1134.387,66.310,-53.199,-179.713,6.597,149.124
C02411=1134.392,66.061,-53.182,-179.716,6.595,149.125
C02412=1134.397,65.811,-53.167,-179.719,6.595,149.125
C02413=1134.402,65.562,-53.150,-179.722,6.593,149.126
C02414=1134.407,65.313,-53.134,-179.724,6.592,149.126
C02415=1134.412,65.063,-53.118,-179.726,6.591,149.127
C02416=1134.417,64.814,-53.101,-179.730,6.590,149.127
C02417=1134.422,64.564,-53.085,-179.732,6.588,149.128
C02418=1134.426,64.314,-53.069,-179.735,6.586,149.128
C02419=1134.432,64.065,-53.052,-179.737,6.585,149.129
C02420=1134.437,63.815,-53.036,-179.741,6.584,149.129
C02421=1134.442,63.567,-53.020,-179.743,6.582,149.130
C02422=1134.447,63.317,-53.004,-179.745,6.582,149.130
C02423=1134.452,63.068,-52.987,-179.748,6.580,149.131
C02424=1134.457,62.818,-52.972,-179.751,6.579,149.131
C02425=1134.462,62.569,-52.955,-179.754,6.578,149.132
C02426=1134.467,62.319,-52.939,-179.756,6.576,149.132
C02427=1134.471,62.070,-52.923,-179.759,6.575,149.133
C02428=1134.477,61.820,-52.907,-179.762,6.574,149.133
C02429=1134.481,61.571,-52.891,-179.765,6.572,149.134
C02430=1134.487,61.322,-52.875,-179.767,6.571,149.134
C02431=1134.491,61.072,-52.858,-179.770,6.570,149.135
C02432=1134.497,60.823,-52.843,-179.773,6.569,149.135
C02433=1134.501,60.573,-52.826,-179.775,6.567,149.136
C02434=1134.506,60.324,-52.810,-179.778,6.566,149.136
C02435=1134.511,60.075,-52.794,-179.781,6.565,149.137
C02436=1134.516,59.825,-52.778,-179.784,6.563,149.137
C02437=1134.522,59.576,-52.763,-179.786,6.563,149.138
C02438=1134.526,59.326,-52.746,-179.788,6.561,149.138
C02439=1134.531,59.077,-52.730,-179.791,6.560,149.139
C02440=1134.537,58.828,-52.714,-179.794,6.559,149.139
C02441=1134.541,58.578,-52.698,-179.797,6.557,149.140
C02442=1134.547,58.328,-52.682,-179.799,6.556,149.140
C02443=1134.551,58.079,-52.666,-179.802,6.555,149.141
C02444=1134.557,57.829,-52.650,-179.805,6.553,149.141
C02445=1134.562,57.580,-52.635,-179.807,6.553,149.142
C02446=1134.566,57.331,-52.618,-179.810,6.551,149.142
C02447=1134.571,57.081,-52.603,-179.813,6.550,149.143
C02448=1134.576,56.831,-52.587,-179.815,6.549,149.143
C02449=1134.581,56.583,-52.571,-179.818,6.547,149.144
C02450=1134.586,56.333,-52.555,-179.820,6.547,149.144
C02451=1134.591,56.083,-52.539,-179.823,6.545,149.145
C02452=1134.597,55.834,-52.524,-179.826,6.543,149.145
C02453=1134.602,55.585,-52.507,-179.828,6.543,149.146
C02454=1134.606,55.335,-52.491,-179.831,6.541,149.146
C02455=1134.612,55.085,-52.476,-179.834,6.540,149.147
C02456=1134.616,54.836,-52.461,-179.836,6.539,149.147
C02457=1134.621,54.586,-52.445,-179.840,6.538,149.148
C02458=1134.626,54.337,-52.428,-179.842,6.537,149.148
C02459=1134.632,54.088,-52.413,-179.844,6.535,149.149
C02460=1134.636,53.838,-52.397,-179.847,6.533,149.149
C02461=1134.642,53.569,-52.380,-179.850,6.533,149.150
C02462=1134.647,53.301,-52.364,-179.853,6.531,149.150
C02463=1134.652,53.033,-52.346,-179.856,6.530,149.151
C02464=1134.658,52.764,-52.330,-179.859,6.529,149.151
C02465=1134.663,52.515,-52.314,-179.861,6.528,149.152
C02466=1134.668,52.265,-52.298,-179.864,6.526,149.153
C02467=1134.673,52.016,-52.283,-179.867,6.525,149.153
C02468=1134.678,51.766,-52.267,-179.869,6.524,149.153
C02469=1134.683,51.516,-52.251,-179.872,6.523,149.154
C02470=1134.688,51.267,-52.236,-179.874,6.522,149.155
C02471=1134.693,51.018,-52.221,-179.877,6.520,149.155
C02472=1134.698,50.768,-52.205,-179.880,6.520,149.156
C02473=1134.703,50.518,-52.189,-179.882,6.518,149.156
C02474=1134.709,50.269,-52.174,-179.885,6.516,149.157
C02475=1134.713,50.020,-52.159,-179.887,6.516,149.157
C02476=1134.719,49.770,-52.143,-179.891,6.514,149.158
C02477=1134.723,49.520,-52.127,-179.893,6.514,149.158
C02478=1134.728,49.271,-52.112,-179.896,6.512,149.159
C02479=1134.733,49.022,-52.097,-179.899,6.511,149.159
C02480=1134.739,48.772,-52.081,-179.901,6.510,149.160
C02481=1134.743,48.523,-52.066,-179.904,6.508,149.160
C02482=1134.748,48.273,-52.050,-179.906,6.507,149.161
C02483=1134.754,48.024,-52.034,-179.909,6.506,149.161
C02484=1134.758,47.775,-52.019,-179.911,6.505,149.162
C02485=1134.764,47.525,-52.004,-179.914,6.504,149.162
C02486=1134.768,47.275,-51.988,-179.917,6.503,149.163
C02487=1134.773,47.026,-51.973,-179.919,6.502,149.163
C02488=1134.778,46.777,-51.957,-179.922,6.500,149.164
C02489=1134.783,46.528,-51.942,-179.925,6.499,149.164
C02490=1134.789,46.278,-51.927,-179.928,6.498,149.165
C02491=1134.794,46.028,-51.912,-179.930,6.497,149.165
C02492=1134.798,45.778,-51.897,-179.933,6.495,149.166
C02493=1134.804,45.529,-51.881,-179.935,6.495,149.166
C02494=1134.808,45.280,-51.866,-179.938,6.493,149.167
C02495=1134.814,45.030,-51.850,-179.940,6.492,149.167
C02496=1134.819,44.781,-51.835,-179.943,6.491,149.168
C02497=1134.824,44.531,-51.820,-179.946,6.490,149.168
C02498=1134.829,44.281,-51.805,-179.948,6.489,149.169
C02499=1134.833,44.032,-51.790,-179.952,6.488,149.169
C02500=1134.839,43.783,-51.774,-179.954,6.487,149.170
C02501=1134.844,43.534,-51.759,-179.956,6.485,149.170
C02502=1134.849,43.284,-51.744,-179.959,6.484,149.171
C02503=1134.854,43.034,-51.729,-179.962,6.483,149.172
C02504=1134.859,42.785,-51.714,-179.964,6.482,149.172
C02505=1134.864,42.536,-51.699,-179.967,6.481,149.172
C02506=1134.869,42.285,-51.683,-179.969,6.480,149.173
C02507=1134.874,42.036,-51.668,-179.972,6.478,149.174
C02508=1134.879,41.787,-51.653,-179.974,6.478,149.174
C02509=1134.884,41.537,-51.638,-179.978,6.476,149.175
C02510=1134.889,41.288,-51.623,-179.980,6.476,149.175
C02511=1134.894,41.039,-51.608,-179.983,6.474,149.176
C02512=1134.900,40.789,-51.593,-179.985,6.473,149.176
C02513=1134.904,40.539,-51.578,-179.988,6.472,149.177
C02514=1134.910,40.290,-51.562,-179.990,6.471,149.177
C02515=1134.915,40.040,-51.548,-179.993,6.470,149.178
C02516=1134.920,39.791,-51.533,-179.995,6.469,149.178
C02517=1134.925,39.542,-51.518,-179.998,6.467,149.179
C02518=1134.930,39.292,-51.503,180.000,6.466,149.179
C02519=1134.935,39.043,-51.488,179.996,6.465,149.180
C02520=1134.940,38.793,-51.473,179.994,6.464,149.180
C02521=1134.945,38.543,-51.457,179.991,6.463,149.181
C02522=1134.949,38.294,-51.442,179.989,6.462,149.181
C02523=1134.954,38.044,-51.428,179.986,6.461,149.182
C02524=1134.960,37.795,-51.413,179.984,6.460,149.182
C02525=1134.965,37.545,-51.398,179.981,6.459,149.183
C02526=1134.970,37.296,-51.383,179.978,6.458,149.183
C02527=1134.975,37.046,-51.368,179.976,6.456,149.184
C02528=1134.980,36.797,-51.353,179.973,6.456,149.185
C02529=1134.985,36.547,-51.339,179.970,6.454,149.185
C02530=1134.990,36.298,-51.324,179.968,6.453,149.185
C02531=1134.995,36.048,-51.309,179.965,6.452,149.186
C02532=1135.000,35.799,-51.294,179.963,6.451,149.187
C02533=1135.005,35.549,-51.279,179.960,6.450,149.187
C02534=1135.010,35.300,-51.264,179.957,6.449,149.188
C02535=1135.016,35.050,-51.250,179.954,6.448,149.188
C02536=1135.021,34.801,-51.235,179.952,6.447,149.189
C02537=1135.026,34.552,-51.221,179.950,6.446,149.189
C02538=1135.032,34.302,-51.206,179.947,6.445,149.190
C02539=1135.036,34.053,-51.191,179.945,6.444,149.190
C02540=1135.041,33.803,-51.177,179.942,6.442,149.191
C02541=1135.046,33.554,-51.162,179.939,6.442,149.191
C02542=1135.052,33.304,-51.147,179.937,6.440,149.192
C02543=1135.057,33.054,-51.132,179.934,6.439,149.192
C02544=1135.061,32.805,-51.117,179.931,6.438,149.193
C02545=1135.066,32.555,-51.103,179.929,6.437,149.193
C02546=1135.072,32.305,-51.088,179.926,6.436,149.194
C02547=1135.076,32.056,-51.073,179.924,6.435,149.194
C02548=1135.081,31.806,-51.059,179.921,6.434,149.195
C02549=1135.086,31.557,-51.045,179.919,6.433,149.195
C02550=1135.092,31.307,-51.029,179.916,6.432,149.196
C02551=1135.097,31.058,-51.015,179.913,6.431,149.196
C02552=1135.102,30.809,-51.001,179.911,6.430,149.197
C02553=1135.107,30.559,-50.986,179.908,6.429,149.198
C02554=1135.112,30.310,-50.972,179.906,6.428,149.198
C02555=1135.117,30.060,-50.957,179.903,6.426,149.199
C02556=1135.123,29.810,-50.943,179.900,6.426,149.199
C02557=1135.127,29.561,-50.928,179.898,6.425,149.200
C02558=1135.132,29.311,-50.913,179.895,6.423,149.200
C02559=1135.137,29.062,-50.899,179.893,6.423,149.201
C02560=1135.143,28.813,-50.885,179.890,6.421,149.201
C02561=1135.148,28.563,-50.871,179.888,6.420,149.202
C02562=1135.153,28.313,-50.855,179.884,6.419,149.202
C02563=1135.158,28.064,-50.841,179.882,6.418,149.203
C02564=1135.163,27.814,-50.827,179.880,6.417,149.203
C02565=1135.168,27.545,-50.811,179.877,6.416,149.204
C02566=1135.173,27.276,-50.796,179.874,6.415,149.204
C02567=1135.179,27.008,-50.781,179.871,6.414,149.205
C02568=1135.185,26.738,-50.765,179.869,6.413,149.206
C02569=1135.190,26.489,-50.750,179.866,6.412,149.206
C02570=1135.195,26.239,-50.736,179.863,6.411,149.207
C02571=1135.200,25.989,-50.721,179.861,6.410,149.207
C02572=1135.205,25.740,-50.707,179.858,6.409,149.208
C02573=1135.210,25.491,-50.693,179.856,6.408,149.208
C02574=1135.215,25.241,-50.679,179.854,6.407,149.209
C02575=1135.220,24.991,-50.665,179.850,6.406,149.209
C02576=1135.225,24.742,-50.650,179.848,6.405,149.210
C02577=1135.230,24.492,-50.636,179.846,6.404,149.210
C02578=1135.236,24.243,-50.622,179.843,6.403,149.211
C02579=1135.241,23.993,-50.608,179.841,6.402,149.211
C02580=1135.246,23.743,-50.594,179.838,6.400,149.212
C02581=1135.251,23.494,-50.579,179.835,6.400,149.213
C02582=1135.256,23.244,-50.565,179.833,6.399,149.213
C02583=1135.261,22.995,-50.551,179.830,6.397,149.214
C02584=1135.266,22.745,-50.537,179.828,6.397,149.214
C02585=1135.271,22.496,-50.523,179.825,6.395,149.215
C02586=1135.276,22.246,-50.508,179.822,6.395,149.215
C02587=1135.282,21.997,-50.494,179.820,6.394,149.216
C02588=1135.287,21.747,-50.480,179.817,6.393,149.216
C02589=1135.292,21.497,-50.466,179.814,6.392,149.217
C02590=1135.296,21.248,-50.452,179.812,6.391,149.217
C02591=1135.302,20.999,-50.438,179.810,6.390,149.218
C02592=1135.307,20.749,-50.423,179.807,6.389,149.219
C02593=1135.312,20.499,-50.409,179.805,6.388,149.219
C02594=1135.317,20.250,-50.395,179.802,6.387,149.219
C02595=1135.322,20.001,-50.381,179.799,6.386,149.220
C02596=1135.327,19.751,-50.367,179.797,6.385,149.221
C02597=1135.332,19.501,-50.354,179.794,6.384,149.221
C02598=1135.337,19.252,-50.340,179.792,6.383,149.222
C02599=1135.342,19.002,-50.326,179.789,6.382,149.222
C02600=1135.347,18.752,-50.311,179.787,6.381,149.223
C02601=1135.353,18.503,-50.297,179.784,6.381,149.223
C02602=1135.358,18.254,-50.283,179.781,6.379,149.224
C02603=1135.363,18.003,-50.270,179.779,6.378,149.224
C02604=1135.369,17.754,-50.256,179.777,6.378,149.225
C02605=1135.373,17.505,-50.242,179.774,6.376,149.225
C02606=1135.378,17.255,-50.228,179.772,6.375,149.226
C02607=1135.383,17.006,-50.214,179.769,6.375,149.227
C02608=1135.389,16.756,-50.200,179.766,6.373,149.227
C02609=1135.394,16.506,-50.186,179.764,6.372,149.227
C02610=1135.399,16.257,-50.172,179.761,6.372,149.228
C02611=1135.403,16.008,-50.158,179.759,6.370,149.229
C02612=1135.409,15.757,-50.145,179.756,6.370,149.229
C02613=1135.414,15.508,-50.131,179.754,6.369,149.230
C02614=1135.419,15.259,-50.117,179.751,6.368,149.230
C02615=1135.424,15.009,-50.102,179.749,6.367,149.231
C02616=1135.429,14.760,-50.090,179.746,6.366,149.231
C02617=1135.434,14.510,-50.075,179.743,6.365,149.232
C02618=1135.440,14.261,-50.062,179.741,6.364,149.232
C02619=1135.445,14.011,-50.048,179.739,6.363,149.233
C02620=1135.449,13.761,-50.034,179.736,6.362,149.233
C02621=1135.455,13.512,-50.020,179.733,6.361,149.234
C02622=1135.460,13.262,-50.007,179.731,6.361,149.235
C02623=1135.466,13.013,-49.993,179.728,6.359,149.235
C02624=1135.470,12.764,-49.979,179.726,6.359,149.236
C02625=1135.475,12.513,-49.966,179.723,6.358,149.236
C02626=1135.481,12.264,-49.952,179.721,6.356,149.237
C02627=1135.486,12.014,-49.938,179.718,6.356,149.237
C02628=1135.491,11.765,-49.925,179.716,6.355,149.238
C02629=1135.496,11.515,-49.911,179.713,6.353,149.238
C02630=1135.502,11.266,-49.897,179.710,6.353,149.239
C02631=1135.506,11.016,-49.884,179.708,6.352,149.239
C02632=1135.511,10.766,-49.870,179.706,6.351,149.240
C02633=1135.517,10.517,-49.856,179.703,6.350,149.241
C02634=1135.521,10.267,-49.843,179.701,6.349,149.241
C02635=1135.527,10.018,-49.829,179.698,6.348,149.241
C02636=1135.532,9.768,-49.816,179.695,6.347,149.242
C02637=1135.537,9.519,-49.802,179.693,6.346,149.243
C02638=1135.542,9.269,-49.789,179.691,6.346,149.243
C02639=1135.548,9.020,-49.775,179.688,6.345,149.244
C02640=1135.552,8.770,-49.762,179.685,6.344,149.244
C02641=1135.558,8.521,-49.748,179.683,6.343,149.245
C02642=1135.563,8.270,-49.735,179.681,6.342,149.245
C02643=1135.568,8.022,-49.721,179.678,6.341,149.246
C02644=1135.573,7.771,-49.708,179.675,6.340,149.246
C02645=1135.578,7.523,-49.694,179.673,6.340,149.247
C02646=1135.583,7.272,-49.681,179.671,6.339,149.247
C02647=1135.589,7.023,-49.668,179.667,6.337,149.248
C02648=1135.593,6.773,-49.654,179.665,6.337,149.249
C02649=1135.599,6.524,-49.641,179.663,6.336,149.249
C02650=1135.603,6.274,-49.627,179.660,6.335,149.250
C02651=1135.609,6.025,-49.614,179.658,6.334,149.250
C02652=1135.614,5.775,-49.601,179.656,6.333,149.251
C02653=1135.619,5.526,-49.587,179.653,6.333,149.251
C02654=1135.624,5.275,-49.573,179.650,6.331,149.252
C02655=1135.629,5.027,-49.560,179.648,6.330,149.252
C02656=1135.634,4.776,-49.547,179.645,6.330,149.253
C02657=1135.640,4.527,-49.534,179.643,6.329,149.253
C02658=1135.645,4.277,-49.520,179.640,6.327,149.254
C02659=1135.650,4.028,-49.507,179.638,6.327,149.255
C02660=1135.656,3.778,-49.494,179.635,6.326,149.255
C02661=1135.660,3.528,-49.481,179.633,6.325,149.255
C02662=1135.666,3.279,-49.467,179.630,6.324,149.256
C02663=1135.670,3.029,-49.454,179.628,6.323,149.257
C02664=1135.676,2.780,-49.441,179.625,6.323,149.257
C02665=1135.680,2.530,-49.427,179.623,6.322,149.258
C02666=1135.686,2.281,-49.414,179.620,6.320,149.258
C02667=1135.691,2.031,-49.401,179.618,6.320,149.259
C02668=1135.696,1.781,-49.388,179.615,6.319,149.259
C02669=1135.701,1.512,-49.373,179.613,6.318,149.260
C02670=1135.708,1.242,-49.359,179.610,6.317,149.261
C02671=1135.713,0.973,-49.346,179.607,6.317,149.261
C02672=1135.718,0.703,-49.331,179.605,6.315,149.262
C02673=1135.723,0.454,-49.318,179.602,6.314,149.262
C02674=1135.729,0.204,-49.305,179.600,6.314,149.263
C02675=1135.733,-0.046,-49.292,179.598,6.313,149.263
C02676=1135.739,-0.295,-49.279,179.595,6.312,149.264
C02677=1135.744,-0.545,-49.265,179.592,6.311,149.265
C02678=1135.749,-0.794,-49.252,179.590,6.310,149.265
C02679=1135.755,-1.044,-49.239,179.587,6.310,149.266
C02680=1135.759,-1.294,-49.226,179.584,6.308,149.266
C02681=1135.765,-1.543,-49.213,179.582,6.308,149.267
C02682=1135.770,-1.793,-49.201,179.580,6.307,149.267
C02683=1135.775,-2.043,-49.188,179.577,6.306,149.268
C02684=1135.780,-2.292,-49.174,179.575,6.306,149.268
C02685=1135.785,-2.541,-49.161,179.572,6.304,149.269
C02686=1135.791,-2.791,-49.148,179.570,6.304,149.269
C02687=1135.796,-3.041,-49.135,179.568,6.303,149.270
C02688=1135.801,-3.290,-49.122,179.565,6.302,149.271
C02689=1135.806,-3.540,-49.109,179.563,6.302,149.271
C02690=1135.811,-3.790,-49.096,179.560,6.300,149.271
C02691=1135.816,-4.039,-49.084,179.557,6.299,149.272
C02692=1135.821,-4.289,-49.071,179.555,6.299,149.273
C02693=1135.827,-4.539,-49.057,179.553,6.298,149.273
C02694=1135.832,-4.788,-49.045,179.550,6.297,149.274
C02695=1135.837,-5.037,-49.032,179.548,6.296,149.274
C02696=1135.842,-5.288,-49.019,179.545,6.295,149.275
C02697=1135.847,-5.537,-49.006,179.543,6.295,149.275
C02698=1135.852,-5.786,-48.993,179.541,6.294,149.276
C02699=1135.857,-6.036,-48.980,179.538,6.293,149.277
C02700=1135.863,-6.286,-48.967,179.535,6.292,149.277
C02701=1135.868,-6.535,-48.955,179.533,6.291,149.277
C02702=1135.873,-6.784,-48.942,179.530,6.291,149.278
C02703=1135.878,-7.034,-48.929,179.528,6.290,149.279
C02704=1135.883,-7.284,-48.916,179.526,6.289,149.279
C02705=1135.889,-7.534,-48.904,179.523,6.289,149.280
C02706=1135.894,-7.783,-48.891,179.521,6.287,149.280
C02707=1135.898,-8.033,-48.878,179.518,6.286,149.281
C02708=1135.904,-8.283,-48.865,179.516,6.286,149.281
C02709=1135.909,-8.532,-48.853,179.514,6.285,149.282
C02710=1135.915,-8.782,-48.840,179.511,6.284,149.282
C02711=1135.919,-9.032,-48.827,179.509,6.284,149.283
C02712=1135.924,-9.281,-48.815,179.506,6.282,149.284
C02713=1135.930,-9.531,-48.801,179.504,6.281,149.284
C02714=1135.936,-9.781,-48.789,179.501,6.281,149.285
C02715=1135.940,-10.031,-48.776,179.499,6.280,149.285
C02716=1135.945,-10.280,-48.764,179.497,6.279,149.286
C02717=1135.950,-10.529,-48.751,179.494,6.279,149.286
C02718=1135.955,-10.778,-48.739,179.491,6.277,149.287
C02719=1135.961,-11.028,-48.727,179.489,6.277,149.287
C02720=1135.966,-11.279,-48.713,179.486,6.276,149.288
C02721=1135.971,-11.528,-48.701,179.484,6.275,149.288
C02722=1135.976,-11.777,-48.688,179.482,6.275,149.289
C02723=1135.981,-12.027,-48.675,179.479,6.274,149.290
C02724=1135.987,-12.277,-48.664,179.477,6.273,149.290
C02725=1135.992,-12.526,-48.651,179.474,6.272,149.291
C02726=1135.997,-12.776,-48.638,179.472,6.271,149.291
C02727=1136.002,-13.025,-48.625,179.470,6.271,149.292
C02728=1136.008,-13.276,-48.613,179.467,6.270,149.292
C02729=1136.013,-13.525,-48.600,179.465,6.269,149.293
C02730=1136.018,-13.774,-48.588,179.463,6.269,149.293
C02731=1136.024,-14.024,-48.576,179.460,6.268,149.294
C02732=1136.028,-14.274,-48.563,179.457,6.267,149.294
C02733=1136.033,-14.523,-48.550,179.455,6.266,149.295
C02734=1136.039,-14.773,-48.538,179.452,6.265,149.296
C02735=1136.044,-15.023,-48.526,179.450,6.265,149.296
C02736=1136.049,-15.272,-48.513,179.448,6.264,149.297
C02737=1136.054,-15.522,-48.501,179.445,6.263,149.297
C02738=1136.059,-15.771,-48.489,179.443,6.263,149.298
C02739=1136.064,-16.021,-48.476,179.441,6.262,149.298
C02740=1136.069,-16.271,-48.464,179.438,6.261,149.299
C02741=1136.074,-16.521,-48.451,179.435,6.260,149.299
C02742=1136.080,-16.770,-48.439,179.433,6.259,149.300
C02743=1136.085,-17.020,-48.427,179.431,6.259,149.301
C02744=1136.090,-17.269,-48.414,179.428,6.258,149.301
C02745=1136.096,-17.519,-48.402,179.426,6.257,149.301
C02746=1136.101,-17.768,-48.390,179.424,6.257,149.302
C02747=1136.106,-18.018,-48.378,179.421,6.256,149.303
C02748=1136.111,-18.268,-48.365,179.419,6.254,149.303
C02749=1136.116,-18.517,-48.353,179.416,6.254,149.304
C02750=1136.121,-18.768,-48.340,179.414,6.253,149.304
C02751=1136.126,-19.017,-48.328,179.411,6.253,149.305
C02752=1136.132,-19.267,-48.316,179.409,6.252,149.305
C02753=1136.137,-19.516,-48.303,179.407,6.251,149.306
C02754=1136.142,-19.766,-48.291,179.404,6.251,149.307
C02755=1136.147,-20.015,-48.279,179.402,6.250,149.307
C02756=1136.153,-20.265,-48.267,179.400,6.249,149.308
C02757=1136.158,-20.515,-48.254,179.397,6.249,149.308
C02758=1136.163,-20.765,-48.242,179.395,6.248,149.309
C02759=1136.169,-21.014,-48.230,179.392,6.246,149.309
C02760=1136.173,-21.264,-48.218,179.389,6.246,149.310
C02761=1136.179,-21.513,-48.207,179.387,6.245,149.310
C02762=1136.184,-21.763,-48.194,179.385,6.244,149.311
C02763=1136.189,-22.013,-48.182,179.382,6.244,149.312
C02764=1136.194,-22.262,-48.169,179.380,6.243,149.312
C02765=1136.200,-22.512,-48.158,179.378,6.242,149.312
C02766=1136.205,-22.761,-48.145,179.375,6.242,149.313
C02767=1136.210,-23.011,-48.133,179.373,6.241,149.314
C02768=1136.216,-23.261,-48.121,179.371,6.240,149.314
C02769=1136.220,-23.510,-48.109,179.368,6.240,149.315
C02770=1136.226,-23.760,-48.097,179.366,6.239,149.315
C02771=1136.231,-24.010,-48.085,179.363,6.238,149.316
C02772=1136.236,-24.259,-48.073,179.361,6.237,149.316
C02773=1136.241,-24.530,-48.060,179.359,6.236,149.317
C02774=1136.247,-24.799,-48.047,179.356,6.236,149.318
C02775=1136.253,-25.070,-48.034,179.354,6.235,149.318
C02776=1136.259,-25.340,-48.021,179.350,6.234,149.319
C02777=1136.263,-25.590,-48.009,179.348,6.233,149.319
C02778=1136.269,-25.839,-47.997,179.346,6.232,149.320
C02779=1136.275,-26.089,-47.985,179.343,6.232,149.320
C02780=1136.280,-26.338,-47.973,179.341,6.231,149.321
C02781=1136.285,-26.588,-47.961,179.339,6.230,149.321
C02782=1136.290,-26.837,-47.950,179.336,6.230,149.322
C02783=1136.295,-27.087,-47.938,179.334,6.229,149.323
C02784=1136.301,-27.337,-47.926,179.332,6.228,149.323
C02785=1136.306,-27.587,-47.913,179.329,6.228,149.324
C02786=1136.310,-27.836,-47.902,179.327,6.227,149.324
C02787=1136.316,-28.086,-47.890,179.325,6.226,149.325
C02788=1136.321,-28.336,-47.878,179.322,6.226,149.325
C02789=1136.326,-28.585,-47.866,179.320,6.225,149.326
C02790=1136.331,-28.835,-47.854,179.318,6.225,149.326
C02791=1136.337,-29.085,-47.842,179.315,6.224,149.327
C02792=1136.342,-29.335,-47.830,179.313,6.223,149.328
C02793=1136.347,-29.585,-47.819,179.311,6.223,149.328
C02794=1136.352,-29.833,-47.807,179.308,6.222,149.329
C02795=1136.358,-30.083,-47.795,179.306,6.221,149.329
C02796=1136.363,-30.333,-47.783,179.304,6.221,149.330
C02797=1136.368,-30.583,-47.772,179.301,6.220,149.330
C02798=1136.373,-30.833,-47.760,179.299,6.219,149.331
C02799=1136.379,-31.083,-47.748,179.296,6.218,149.331
C02800=1136.383,-31.332,-47.736,179.294,6.217,149.332
C02801=1136.389,-31.582,-47.724,179.291,6.217,149.332
C02802=1136.394,-31.831,-47.712,179.289,6.216,149.333
C02803=1136.399,-32.080,-47.701,179.286,6.215,149.334
C02804=1136.405,-32.330,-47.690,179.284,6.215,149.334
C02805=1136.410,-32.580,-47.678,179.282,6.214,149.335
C02806=1136.415,-32.830,-47.666,179.279,6.213,149.335
C02807=1136.420,-33.080,-47.654,179.277,6.213,149.336
C02808=1136.425,-33.329,-47.643,179.275,6.212,149.336
C02809=1136.430,-33.579,-47.631,179.272,6.212,149.337
C02810=1136.437,-33.829,-47.620,179.270,6.211,149.337
C02811=1136.441,-34.078,-47.608,179.268,6.210,149.338
C02812=1136.447,-34.328,-47.597,179.266,6.209,149.338
C02813=1136.452,-34.578,-47.585,179.263,6.209,149.339
C02814=1136.456,-34.827,-47.573,179.261,6.208,149.340
C02815=1136.462,-35.077,-47.561,179.259,6.207,149.340
C02816=1136.467,-35.326,-47.550,179.256,6.207,149.341
C02817=1136.473,-35.576,-47.538,179.254,6.206,149.341
C02818=1136.477,-35.826,-47.527,179.252,6.205,149.342
C02819=1136.483,-36.076,-47.516,179.249,6.205,149.342
C02820=1136.488,-36.326,-47.504,179.247,6.204,149.343
C02821=1136.494,-36.575,-47.493,179.245,6.203,149.343
C02822=1136.499,-36.825,-47.481,179.242,6.203,149.344
C02823=1136.504,-37.075,-47.470,179.240,6.202,149.344
C02824=1136.509,-37.324,-47.458,179.238,6.201,149.345
C02825=1136.515,-37.573,-47.447,179.235,6.201,149.346
C02826=1136.520,-37.823,-47.435,179.233,6.200,149.346
C02827=1136.525,-38.073,-47.424,179.231,6.199,149.347
C02828=1136.530,-38.323,-47.412,179.228,6.199,149.347
C02829=1136.535,-38.572,-47.400,179.226,6.198,149.348
C02830=1136.541,-38.822,-47.389,179.224,6.197,149.348
C02831=1136.546,-39.071,-47.378,179.221,6.197,149.349
C02832=1136.551,-39.322,-47.366,179.219,6.196,149.349
C02833=1136.556,-39.572,-47.355,179.217,6.196,149.350
C02834=1136.562,-39.821,-47.344,179.215,6.195,149.350
C02835=1136.567,-40.070,-47.332,179.212,6.195,149.351
C02836=1136.572,-40.320,-47.320,179.210,6.194,149.352
C02837=1136.577,-40.570,-47.309,179.208,6.194,149.352
C02838=1136.583,-40.819,-47.298,179.205,6.193,149.353
C02839=1136.588,-41.069,-47.287,179.203,6.192,149.353
C02840=1136.593,-41.319,-47.275,179.201,6.192,149.354
C02841=1136.599,-41.568,-47.264,179.198,6.191,149.354
C02842=1136.604,-41.818,-47.252,179.196,6.190,149.355
C02843=1136.609,-42.068,-47.241,179.194,6.190,149.355
C02844=1136.614,-42.318,-47.230,179.192,6.189,149.356
C02845=1136.620,-42.567,-47.219,179.189,6.188,149.357
C02846=1136.624,-42.817,-47.208,179.187,6.188,149.357
C02847=1136.630,-43.067,-47.196,179.185,6.187,149.357
C02848=1136.635,-43.316,-47.186,179.182,6.187,149.358
C02849=1136.641,-43.566,-47.174,179.180,6.186,149.359
C02850=1136.646,-43.816,-47.162,179.178,6.185,149.359
C02851=1136.651,-44.065,-47.152,179.175,6.185,149.360
C02852=1136.657,-44.315,-47.140,179.173,6.184,149.360
C02853=1136.661,-44.565,-47.129,179.171,6.183,149.361
C02854=1136.667,-44.814,-47.118,179.168,6.183,149.361
C02855=1136.672,-45.065,-47.107,179.166,6.182,149.362
C02856=1136.677,-45.314,-47.096,179.164,6.182,149.362
C02857=1136.683,-45.563,-47.084,179.162,6.181,149.363
C02858=1136.688,-45.813,-47.073,179.159,6.181,149.364
C02859=1136.693,-46.063,-47.062,179.157,6.180,149.364
C02860=1136.699,-46.313,-47.051,179.155,6.179,149.365
C02861=1136.703,-46.562,-47.039,179.152,6.179,149.365
C02862=1136.708,-46.812,-47.029,179.150,6.178,149.366
C02863=1136.714,-47.062,-47.017,179.148,6.177,149.366
C02864=1136.719,-47.312,-47.007,179.146,6.176,149.367
C02865=1136.724,-47.562,-46.996,179.143,6.176,149.367
C02866=1136.729,-47.810,-46.985,179.141,6.175,149.368
C02867=1136.735,-48.061,-46.973,179.139,6.174,149.368
C02868=1136.740,-48.311,-46.962,179.136,6.174,149.369
C02869=1136.745,-48.560,-46.952,179.134,6.173,149.370
C02870=1136.751,-48.810,-46.940,179.132,6.173,149.370
C02871=1136.756,-49.059,-46.929,179.130,6.173,149.371
C02872=1136.761,-49.309,-46.919,179.127,6.172,149.371
C02873=1136.767,-49.559,-46.907,179.125,6.171,149.372
C02874=1136.772,-49.809,-46.896,179.123,6.171,149.372
C02875=1136.777,-50.058,-46.885,179.120,6.170,149.373
C02876=1136.783,-50.308,-46.875,179.118,6.169,149.373
C02877=1136.788,-50.579,-46.863,179.116,6.169,149.374
C02878=1136.794,-50.850,-46.850,179.113,6.168,149.375
C02879=1136.800,-51.120,-46.839,179.111,6.168,149.375
C02880=1136.805,-51.391,-46.827,179.108,6.167,149.376
C02881=1136.811,-51.641,-46.816,179.106,6.166,149.376
C02882=1136.816,-51.890,-46.805,179.104,6.166,149.377
C02883=1136.821,-52.141,-46.794,179.101,6.165,149.377
C02884=1136.826,-52.389,-46.783,179.099,6.164,149.378
C02885=1136.831,-52.640,-46.773,179.097,6.164,149.378
C02886=1136.837,-52.889,-46.761,179.094,6.163,149.379
C02887=1136.842,-53.139,-46.751,179.092,6.163,149.380
C02888=1136.848,-53.389,-46.740,179.090,6.163,149.380
C02889=1136.852,-53.638,-46.729,179.088,6.162,149.380
C02890=1136.858,-53.888,-46.719,179.086,6.161,149.381
C02891=1136.863,-54.138,-46.708,179.083,6.161,149.382
C02892=1136.869,-54.388,-46.696,179.081,6.160,149.382
C02893=1136.874,-54.637,-46.686,179.079,6.159,149.383
C02894=1136.879,-54.887,-46.675,179.076,6.159,149.383
C02895=1136.884,-55.137,-46.665,179.074,6.158,149.384
C02896=1136.889,-55.386,-46.653,179.073,6.158,149.384
C02897=1136.895,-55.636,-46.643,179.070,6.158,149.385
C02898=1136.899,-55.886,-46.632,179.068,6.157,149.385
C02899=1136.906,-56.135,-46.621,179.066,6.156,149.386
C02900=1136.911,-56.386,-46.611,179.063,6.155,149.386
C02901=1136.916,-56.635,-46.600,179.061,6.155,149.387
C02902=1136.921,-56.885,-46.589,179.058,6.154,149.388
C02903=1136.927,-57.134,-46.579,179.056,6.153,149.388
C02904=1136.931,-57.384,-46.568,179.055,6.153,149.389
C02905=1136.937,-57.634,-46.557,179.052,6.153,149.389
C02906=1136.942,-57.884,-46.547,179.050,6.152,149.390
C02907=1136.947,-58.133,-46.536,179.048,6.151,149.390
C02908=1136.952,-58.383,-46.525,179.045,6.151,149.391
C02909=1136.958,-58.633,-46.515,179.043,6.150,149.391
C02910=1136.963,-58.883,-46.505,179.041,6.149,149.392
C02911=1136.969,-59.132,-46.493,179.038,6.149,149.392
C02912=1136.974,-59.382,-46.482,179.036,6.149,149.393
C02913=1136.979,-59.632,-46.472,179.034,6.148,149.394
C02914=1136.984,-59.881,-46.461,179.032,6.148,149.394
C02915=1136.990,-60.131,-46.451,179.030,6.147,149.395
C02916=1136.995,-60.381,-46.441,179.027,6.146,149.395
C02917=1137.000,-60.631,-46.430,179.025,6.146,149.396
C02918=1137.006,-60.880,-46.420,179.023,6.146,149.396
C02919=1137.011,-61.130,-46.408,179.021,6.145,149.397
C02920=1137.016,-61.379,-46.398,179.018,6.145,149.397
C02921=1137.021,-61.630,-46.388,179.016,6.144,149.398
C02922=1137.027,-61.879,-46.377,179.014,6.143,149.398
C02923=1137.032,-62.129,-46.367,179.012,6.142,149.399
C02924=1137.037,-62.378,-46.356,179.009,6.142,149.400
C02925=1137.043,-62.628,-46.346,179.008,6.142,149.400
C02926=1137.048,-62.878,-46.335,179.005,6.141,149.400
C02927=1137.053,-63.128,-46.325,179.003,6.140,149.401
C02928=1137.058,-63.378,-46.314,179.001,6.140,149.402
C02929=1137.064,-63.628,-46.304,178.998,6.139,149.402
C02930=1137.069,-63.876,-46.293,178.996,6.138,149.403
C02931=1137.074,-64.127,-46.283,178.995,6.138,149.403
C02932=1137.079,-64.376,-46.273,178.992,6.138,149.404
C02933=1137.084,-64.626,-46.263,178.990,6.137,149.404
C02934=1137.090,-64.876,-46.252,178.988,6.137,149.405
C02935=1137.095,-65.125,-46.242,178.985,6.136,149.405
C02936=1137.100,-65.376,-46.232,178.983,6.135,149.406
C02937=1137.106,-65.625,-46.221,178.981,6.135,149.406
C02938=1137.111,-65.875,-46.211,178.979,6.135,149.407
C02939=1137.116,-66.125,-46.201,178.977,6.134,149.407
C02940=1137.122,-66.374,-46.190,178.974,6.134,149.408
C02941=1137.127,-66.623,-46.179,178.972,6.133,149.409
C02942=1137.132,-66.874,-46.169,178.970,6.133,149.409
C02943=1137.138,-67.123,-46.159,178.968,6.132,149.410
C02944=1137.142,-67.373,-46.149,178.965,6.132,149.410
C02945=1137.148,-67.623,-46.138,178.963,6.131,149.411
C02946=1137.153,-67.872,-46.128,178.961,6.130,149.411
C02947=1137.158,-68.122,-46.118,178.959,6.130,149.412
C02948=1137.164,-68.372,-46.107,178.957,6.130,149.412
C02949=1137.170,-68.621,-46.097,178.955,6.129,149.413
C02950=1137.175,-68.872,-46.087,178.952,6.128,149.413
C02951=1137.180,-69.121,-46.076,178.950,6.127,149.414
C02952=1137.185,-69.370,-46.067,178.949,6.127,149.414
C02953=1137.191,-69.620,-46.057,178.946,6.127,149.415
C02954=1137.196,-69.870,-46.046,178.944,6.126,149.416
C02955=1137.201,-70.120,-46.036,178.942,6.126,149.416
C02956=1137.207,-70.370,-46.026,178.939,6.125,149.417
C02957=1137.212,-70.620,-46.016,178.937,6.125,149.417
C02958=1137.217,-70.869,-46.006,178.935,6.124,149.418
C02959=1137.223,-71.119,-45.996,178.933,6.124,149.418
C02960=1137.228,-71.369,-45.985,178.931,6.123,149.419
C02961=1137.233,-71.619,-45.975,178.928,6.123,149.419
C02962=1137.239,-71.868,-45.965,178.926,6.123,149.420
C02963=1137.244,-72.118,-45.955,178.924,6.122,149.420
C02964=1137.249,-72.368,-45.945,178.922,6.121,149.421
C02965=1137.254,-72.617,-45.935,178.920,6.120,149.421
C02966=1137.260,-72.867,-45.924,178.917,6.120,149.422
C02967=1137.266,-73.117,-45.915,178.916,6.120,149.422
C02968=1137.270,-73.367,-45.905,178.913,6.119,149.423
C02969=1137.276,-73.617,-45.895,178.911,6.118,149.423
C02970=1137.281,-73.866,-45.884,178.909,6.118,149.424
C02971=1137.287,-74.116,-45.874,178.907,6.118,149.425
C02972=1137.291,-74.366,-45.864,178.905,6.117,149.425
C02973=1137.297,-74.616,-45.855,178.903,6.117,149.426
C02974=1137.303,-74.865,-45.845,178.900,6.116,149.426
C02975=1137.308,-75.115,-45.834,178.898,6.115,149.427
C02976=1137.312,-75.365,-45.824,178.896,6.115,149.427
C02977=1137.318,-75.614,-45.814,178.894,6.115,149.428
C02978=1137.324,-75.864,-45.805,178.892,6.114,149.428
C02979=1137.329,-76.114,-45.795,178.889,6.113,149.429
C02980=1137.334,-76.363,-45.785,178.887,6.114,149.429
C02981=1137.340,-76.635,-45.773,178.885,6.113,149.430
C02982=1137.346,-76.907,-45.763,178.883,6.112,149.430
C02983=1137.351,-77.178,-45.752,178.880,6.112,149.431
C02984=1137.358,-77.450,-45.742,178.878,6.111,149.432
C02985=1137.363,-77.700,-45.731,178.876,6.110,149.432
C02986=1137.368,-77.949,-45.722,178.873,6.110,149.433
C02987=1137.373,-78.199,-45.711,178.872,6.110,149.433
C02988=1137.379,-78.449,-45.702,178.870,6.109,149.434
C02989=1137.384,-78.698,-45.692,178.867,6.108,149.434
C02990=1137.390,-78.948,-45.682,178.865,6.108,149.435
C02991=1137.395,-79.198,-45.672,178.863,6.108,149.435
C02992=1137.400,-79.448,-45.663,178.861,6.107,149.436
C02993=1137.405,-79.697,-45.652,178.859,6.106,149.436
C02994=1137.411,-79.947,-45.643,178.857,6.107,149.437
C02995=1137.416,-80.197,-45.633,178.855,6.106,149.437
C02996=1137.422,-80.446,-45.623,178.852,6.105,149.438
C02997=1137.426,-80.697,-45.614,178.850,6.105,149.439
C02998=1137.432,-80.946,-45.604,178.848,6.105,149.439
C02999=1137.437,-81.196,-45.593,178.846,6.104,149.440
C03000=1137.443,-81.446,-45.584,178.844,6.103,149.440
C03001=1137.448,-81.695,-45.574,178.841,6.103,149.441
C03002=1137.453,-81.944,-45.565,178.840,6.103,149.441
C03003=1137.459,-82.195,-45.555,178.838,6.102,149.442
C03004=1137.464,-82.445,-45.545,178.835,6.101,149.442
C03005=1137.469,-82.695,-45.536,178.833,6.101,149.443
C03006=1137.475,-82.944,-45.525,178.832,6.101,149.443
C03007=1137.480,-83.193,-45.516,178.829,6.100,149.444
C03008=1137.486,-83.444,-45.506,178.827,6.099,149.444
C03009=1137.490,-83.693,-45.497,178.825,6.099,149.445
C03010=1137.496,-83.943,-45.487,178.823,6.099,149.445
C03011=1137.501,-84.192,-45.478,178.821,6.098,149.446
C03012=1137.506,-84.443,-45.468,178.819,6.097,149.446
C03013=1137.512,-84.693,-45.458,178.816,6.098,149.447
C03014=1137.517,-84.942,-45.449,178.814,6.097,149.447
C03015=1137.523,-85.192,-45.438,178.812,6.096,149.448
C03016=1137.528,-85.442,-45.430,178.810,6.096,149.448
C03017=1137.534,-85.691,-45.419,178.808,6.095,149.449
C03018=1137.538,-85.941,-45.410,178.806,6.095,149.450
C03019=1137.544,-86.191,-45.400,178.803,6.094,149.450
C03020=1137.549,-86.440,-45.391,178.802,6.094,149.451
C03021=1137.555,-86.691,-45.381,178.800,6.094,149.451
C03022=1137.560,-86.941,-45.372,178.797,6.093,149.452
C03023=1137.565,-87.190,-45.362,178.796,6.093,149.452
C03024=1137.570,-87.440,-45.353,178.793,6.092,149.453
C03025=1137.575,-87.689,-45.343,178.791,6.092,149.453
C03026=1137.581,-87.940,-45.334,178.789,6.091,149.454
C03027=1137.586,-88.189,-45.324,178.787,6.091,149.454
C03028=1137.592,-88.439,-45.315,178.785,6.090,149.455
C03029=1137.597,-88.688,-45.305,178.783,6.089,149.455
C03030=1137.603,-88.938,-45.295,178.781,6.089,149.456
C03031=1137.608,-89.188,-45.286,178.779,6.089,149.456
C03032=1137.614,-89.438,-45.276,178.776,6.088,149.457
C03033=1137.619,-89.688,-45.267,178.775,6.088,149.457
C03034=1137.624,-89.937,-45.257,178.773,6.088,149.458
C03035=1137.629,-90.187,-45.248,178.770,6.087,149.458
C03036=1137.634,-90.436,-45.239,178.769,6.087,149.459
C03037=1137.640,-90.686,-45.229,178.766,6.087,149.460
C03038=1137.645,-90.936,-45.220,178.764,6.086,149.460
C03039=1137.651,-91.186,-45.210,178.762,6.085,149.460
C03040=1137.656,-91.436,-45.201,178.760,6.085,149.461
C03041=1137.661,-91.685,-45.192,178.758,6.084,149.461
C03042=1137.667,-91.935,-45.182,178.756,6.084,149.462
C03043=1137.672,-92.185,-45.173,178.754,6.084,149.462
C03044=1137.678,-92.435,-45.164,178.751,6.083,149.463
C03045=1137.683,-92.684,-45.154,178.749,6.083,149.464
C03046=1137.688,-92.934,-45.145,178.748,6.083,149.464
C03047=1137.694,-93.184,-45.136,178.745,6.082,149.465
C03048=1137.699,-93.433,-45.126,178.743,6.081,149.465
C03049=1137.704,-93.683,-45.117,178.742,6.081,149.466
C03050=1137.710,-93.934,-45.108,178.739,6.080,149.466
C03051=1137.715,-94.183,-45.098,178.737,6.080,149.467
C03052=1137.720,-94.433,-45.089,178.735,6.080,149.467
C03053=1137.726,-94.683,-45.080,178.733,6.079,149.468
C03054=1137.731,-94.933,-45.071,178.731,6.078,149.468
C03055=1137.736,-95.182,-45.061,178.729,6.079,149.469
C03056=1137.742,-95.432,-45.052,178.727,6.078,149.469
C03057=1137.747,-95.682,-45.043,178.725,6.077,149.470
C03058=1137.752,-95.932,-45.034,178.723,6.077,149.470
C03059=1137.758,-96.181,-45.024,178.721,6.077,149.471
C03060=1137.763,-96.431,-45.015,178.718,6.076,149.471
C03061=1137.768,-96.681,-45.006,178.717,6.076,149.472
C03062=1137.774,-96.931,-44.996,178.715,6.075,149.472
C03063=1137.779,-97.181,-44.987,178.712,6.074,149.473
C03064=1137.784,-97.430,-44.978,178.711,6.075,149.473
C03065=1137.790,-97.680,-44.968,178.709,6.074,149.474
C03066=1137.795,-97.930,-44.959,178.706,6.073,149.474
C03067=1137.800,-98.180,-44.951,178.705,6.073,149.475
C03068=1137.805,-98.430,-44.942,178.702,6.073,149.475
C03069=1137.811,-98.679,-44.932,178.701,6.073,149.476
C03070=1137.817,-98.929,-44.923,178.698,6.072,149.476
C03071=1137.822,-99.178,-44.914,178.696,6.071,149.477
C03072=1137.827,-99.428,-44.905,178.695,6.071,149.477
C03073=1137.833,-99.678,-44.896,178.692,6.071,149.478
C03074=1137.838,-99.928,-44.887,178.690,6.070,149.478
C03075=1137.843,-100.178,-44.878,178.689,6.070,149.479
C03076=1137.848,-100.428,-44.869,178.686,6.069,149.479
C03077=1137.854,-100.678,-44.859,178.684,6.069,149.480
C03078=1137.859,-100.927,-44.850,178.682,6.069,149.481
C03079=1137.865,-101.177,-44.841,178.680,6.068,149.481
C03080=1137.870,-101.426,-44.832,178.678,6.068,149.481
C03081=1137.875,-101.676,-44.824,178.676,6.067,149.482
C03082=1137.881,-101.926,-44.814,178.674,6.067,149.482
C03083=1137.886,-102.176,-44.805,178.672,6.067,149.483
C03084=1137.892,-102.426,-44.796,178.670,6.066,149.483
C03085=1137.897,-102.698,-44.786,178.667,6.065,149.484
C03086=1137.903,-102.971,-44.776,178.665,6.065,149.485
C03087=1137.909,-103.242,-44.767,178.664,6.065,149.485
C03088=1137.915,-103.514,-44.757,178.661,6.064,149.486
C03089=1137.921,-103.765,-44.748,178.659,6.063,149.486
C03090=1137.926,-104.014,-44.739,178.657,6.064,149.487
C03091=1137.931,-104.264,-44.730,178.655,6.063,149.487
C03092=1137.936,-104.514,-44.721,178.653,6.062,149.488
C03093=1137.941,-104.764,-44.712,178.651,6.062,149.488
C03094=1137.947,-105.013,-44.704,178.649,6.061,149.489
C03095=1137.952,-105.263,-44.695,178.647,6.062,149.489
C03096=1137.958,-105.513,-44.685,178.645,6.061,149.490
C03097=1137.963,-105.763,-44.676,178.643,6.060,149.490
C03098=1137.968,-106.013,-44.667,178.641,6.060,149.491
C03099=1137.974,-106.263,-44.658,178.639,6.059,149.491
C03100=1137.979,-106.512,-44.650,178.638,6.059,149.492
C03101=1137.985,-106.762,-44.641,178.635,6.059,149.492
C03102=1137.990,-107.012,-44.632,178.633,6.058,149.493
C03103=1137.995,-107.261,-44.623,178.631,6.058,149.493
C03104=1138.000,-107.511,-44.614,178.629,6.058,149.494
C03105=1138.006,-107.761,-44.606,178.627,6.058,149.494
C03106=1138.012,-108.011,-44.597,178.625,6.057,149.495
C03107=1138.017,-108.261,-44.588,178.623,6.056,149.495
C03108=1138.022,-108.511,-44.579,178.621,6.056,149.496
C03109=1138.028,-108.761,-44.570,178.619,6.055,149.496
C03110=1138.033,-109.010,-44.562,178.618,6.055,149.497
C03111=1138.038,-109.260,-44.553,178.615,6.055,149.497
C03112=1138.044,-109.510,-44.544,178.613,6.054,149.498
C03113=1138.049,-109.759,-44.535,178.612,6.054,149.498
C03114=1138.054,-110.009,-44.526,178.609,6.053,149.499
C03115=1138.060,-110.259,-44.518,178.608,6.053,149.499
C03116=1138.065,-110.509,-44.509,178.606,6.053,149.500
C03117=1138.070,-110.759,-44.501,178.603,6.052,149.500
C03118=1138.076,-111.009,-44.492,178.602,6.052,149.501
C03119=1138.081,-111.258,-44.483,178.599,6.051,149.501
C03120=1138.086,-111.508,-44.474,178.598,6.052,149.502
C03121=1138.092,-111.758,-44.466,178.595,6.051,149.502
C03122=1138.097,-112.008,-44.457,178.594,6.051,149.503
C03123=1138.103,-112.257,-44.449,178.592,6.050,149.503
C03124=1138.108,-112.507,-44.440,178.589,6.049,149.504
C03125=1138.113,-112.757,-44.431,178.588,6.049,149.504
C03126=1138.118,-113.007,-44.422,178.586,6.049,149.505
C03127=1138.124,-113.256,-44.414,178.584,6.049,149.505
C03128=1138.130,-113.506,-44.405,178.582,6.048,149.506
C03129=1138.135,-113.756,-44.396,178.580,6.047,149.506
C03130=1138.141,-114.005,-44.388,178.578,6.047,149.507
C03131=1138.146,-114.256,-44.380,178.576,6.046,149.507
C03132=1138.151,-114.506,-44.371,178.574,6.046,149.508
C03133=1138.156,-114.755,-44.362,178.572,6.046,149.508
C03134=1138.162,-115.005,-44.353,178.570,6.046,149.509
C03135=1138.168,-115.255,-44.345,178.568,6.045,149.509
C03136=1138.173,-115.505,-44.336,178.566,6.044,149.510
C03137=1138.178,-115.754,-44.328,178.564,6.044,149.510
C03138=1138.184,-116.004,-44.319,178.562,6.044,149.511
C03139=1138.189,-116.254,-44.311,178.561,6.044,149.511
C03140=1138.194,-116.504,-44.302,178.558,6.043,149.512
C03141=1138.200,-116.753,-44.293,178.557,6.043,149.512
C03142=1138.206,-117.004,-44.285,178.555,6.042,149.513
C03143=1138.211,-117.254,-44.276,178.553,6.042,149.513
C03144=1138.216,-117.502,-44.268,178.551,6.041,149.514
C03145=1138.221,-117.753,-44.260,178.549,6.041,149.514
C03146=1138.226,-118.003,-44.251,178.547,6.041,149.515
C03147=1138.232,-118.252,-44.243,178.545,6.040,149.515
C03148=1138.238,-118.502,-44.234,178.543,6.040,149.516
C03149=1138.243,-118.752,-44.225,178.541,6.039,149.516
C03150=1138.249,-119.001,-44.217,178.539,6.039,149.516
C03151=1138.254,-119.252,-44.209,178.537,6.039,149.517
C03152=1138.259,-119.502,-44.200,178.536,6.039,149.517
C03153=1138.264,-119.751,-44.192,178.533,6.038,149.518
C03154=1138.270,-120.001,-44.184,178.532,6.038,149.518
C03155=1138.275,-120.251,-44.175,178.530,6.037,149.519
C03156=1138.281,-120.501,-44.167,178.527,6.037,149.519
C03157=1138.286,-120.751,-44.158,178.526,6.037,149.520
C03158=1138.292,-121.000,-44.150,178.524,6.036,149.520
C03159=1138.297,-121.250,-44.141,178.522,6.036,149.521
C03160=1138.302,-121.500,-44.133,178.520,6.035,149.521
C03161=1138.308,-121.749,-44.125,178.518,6.035,149.522
C03162=1138.313,-121.999,-44.116,178.516,6.034,149.522
C03163=1138.318,-122.249,-44.107,178.514,6.034,149.523
C03164=1138.324,-122.499,-44.100,178.512,6.034,149.523
C03165=1138.329,-122.749,-44.091,178.511,6.034,149.524
C03166=1138.334,-122.999,-44.083,178.508,6.033,149.524
C03167=1138.340,-123.248,-44.075,178.507,6.033,149.525
C03168=1138.345,-123.499,-44.066,178.505,6.032,149.525
C03169=1138.351,-123.748,-44.058,178.503,6.032,149.526
C03170=1138.357,-123.998,-44.050,178.501,6.032,149.526
C03171=1138.361,-124.248,-44.041,178.499,6.031,149.527
C03172=1138.367,-124.498,-44.034,178.497,6.031,149.527
C03173=1138.372,-124.747,-44.025,178.495,6.030,149.528
C03174=1138.378,-124.997,-44.017,178.493,6.030,149.528
C03175=1138.383,-125.247,-44.009,178.491,6.029,149.529
C03176=1138.389,-125.496,-44.001,178.489,6.030,149.529
C03177=1138.394,-125.746,-43.992,178.487,6.029,149.530
C03178=1138.400,-125.997,-43.984,178.486,6.029,149.530
C03179=1138.405,-126.246,-43.976,178.483,6.028,149.531
C03180=1138.410,-126.496,-43.968,178.482,6.028,149.531
C03181=1138.416,-126.745,-43.959,178.480,6.027,149.532
C03182=1138.421,-126.996,-43.951,178.478,6.027,149.532
C03183=1138.426,-127.245,-43.943,178.476,6.027,149.533
C03184=1138.432,-127.495,-43.935,178.474,6.027,149.533
C03185=1138.437,-127.745,-43.927,178.472,6.026,149.534
C03186=1138.443,-127.995,-43.918,178.470,6.026,149.534
C03187=1138.448,-128.245,-43.910,178.468,6.025,149.535
C03188=1138.453,-128.494,-43.902,178.467,6.025,149.535
C03189=1138.033,-128.505,-43.945,178.463,6.028,149.537
C03190=1138.027,-128.256,-43.954,178.466,6.029,149.536
C03191=1138.022,-128.006,-43.962,178.467,6.029,149.536
C03192=1138.016,-127.756,-43.970,178.469,6.030,149.535
C03193=1138.011,-127.506,-43.978,178.471,6.030,149.535
C03194=1138.005,-127.257,-43.986,178.473,6.031,149.534
C03195=1138.000,-127.007,-43.995,178.474,6.031,149.534
C03196=1137.994,-126.757,-44.003,178.476,6.031,149.533
C03197=1137.990,-126.507,-44.011,178.478,6.031,149.533
C03198=1137.984,-126.257,-44.019,178.480,6.032,149.532
C03199=1137.978,-126.007,-44.027,178.482,6.032,149.532
C03200=1137.973,-125.757,-44.036,178.484,6.033,149.531
C03201=1137.968,-125.508,-44.043,178.486,6.033,149.531
C03202=1137.962,-125.258,-44.052,178.488,6.034,149.530
C03203=1137.957,-125.008,-44.060,178.489,6.034,149.530
C03204=1137.951,-124.758,-44.069,178.492,6.034,149.530
C03205=1137.946,-124.508,-44.076,178.493,6.034,149.529
C03206=1137.941,-124.259,-44.085,178.495,6.035,149.529
C03207=1137.935,-124.009,-44.093,178.498,6.036,149.528
C03208=1137.929,-123.760,-44.102,178.499,6.036,149.528
C03209=1137.924,-123.509,-44.110,178.501,6.036,149.527
C03210=1137.920,-123.260,-44.118,178.503,6.036,149.527
C03211=1137.914,-123.010,-44.127,178.505,6.037,149.526
C03212=1137.908,-122.760,-44.135,178.507,6.037,149.526
C03213=1137.903,-122.510,-44.144,178.509,6.038,149.525
C03214=1137.897,-122.260,-44.152,178.511,6.038,149.525
C03215=1137.893,-122.011,-44.160,178.513,6.038,149.524
C03216=1137.887,-121.761,-44.168,178.514,6.038,149.524
C03217=1137.881,-121.511,-44.177,178.517,6.039,149.523
C03218=1137.876,-121.261,-44.185,178.518,6.039,149.523
C03219=1137.870,-121.012,-44.193,178.520,6.040,149.522
C03220=1137.865,-120.762,-44.202,178.522,6.040,149.522
C03221=1137.860,-120.511,-44.210,178.524,6.041,149.521
C03222=1137.855,-120.262,-44.218,178.526,6.041,149.521
C03223=1137.849,-120.012,-44.227,178.528,6.041,149.520
C03224=1137.844,-119.762,-44.235,178.530,6.042,149.520
C03225=1137.838,-119.513,-44.244,178.532,6.042,149.519
C03226=1137.833,-119.262,-44.252,178.534,6.043,149.519
C03227=1137.827,-119.013,-44.261,178.536,6.043,149.518
C03228=1137.822,-118.763,-44.270,178.538,6.043,149.518
C03229=1137.817,-118.513,-44.277,178.539,6.043,149.517
C03230=1137.812,-118.263,-44.286,178.542,6.044,149.517
C03231=1137.806,-118.014,-44.295,178.543,6.044,149.516
C03232=1137.801,-117.764,-44.303,178.545,6.045,149.516
C03233=1137.795,-117.514,-44.312,178.548,6.046,149.515
C03234=1137.790,-117.265,-44.320,178.549,6.046,149.515
C03235=1137.784,-117.014,-44.328,178.551,6.046,149.514
C03236=1137.779,-116.764,-44.337,178.553,6.046,149.514
C03237=1137.773,-116.515,-44.346,178.555,6.047,149.513
C03238=1137.768,-116.265,-44.354,178.557,6.047,149.513
C03239=1137.763,-116.015,-44.363,178.559,6.048,149.512
C03240=1137.757,-115.766,-44.371,178.561,6.048,149.512
C03241=1137.752,-115.516,-44.379,178.563,6.048,149.511
C03242=1137.747,-115.266,-44.388,178.565,6.049,149.511
C03243=1137.741,-115.017,-44.396,178.567,6.049,149.511
C03244=1137.736,-114.767,-44.405,178.569,6.050,149.510
C03245=1137.731,-114.516,-44.414,178.570,6.050,149.510
C03246=1137.725,-114.266,-44.422,178.573,6.051,149.509
C03247=1137.720,-114.017,-44.431,178.574,6.050,149.509
C03248=1137.714,-113.767,-44.440,178.576,6.051,149.508
C03249=1137.709,-113.517,-44.448,178.578,6.052,149.508
C03250=1137.703,-113.268,-44.457,178.580,6.052,149.507
C03251=1137.698,-113.018,-44.465,178.582,6.053,149.507
C03252=1137.693,-112.768,-44.474,178.584,6.053,149.506
C03253=1137.688,-112.518,-44.483,178.586,6.053,149.506
C03254=1137.682,-112.269,-44.491,178.588,6.053,149.505
C03255=1137.676,-112.019,-44.500,178.590,6.054,149.505
C03256=1137.671,-111.769,-44.509,178.592,6.055,149.504
C03257=1137.666,-111.519,-44.518,178.594,6.055,149.504
C03258=1137.660,-111.270,-44.526,178.596,6.056,149.503
C03259=1137.655,-111.020,-44.535,178.598,6.055,149.502
C03260=1137.650,-110.770,-44.543,178.600,6.056,149.502
C03261=1137.645,-110.520,-44.552,178.602,6.057,149.502
C03262=1137.639,-110.271,-44.561,178.604,6.057,149.501
C03263=1137.634,-110.021,-44.570,178.606,6.057,149.501
C03264=1137.628,-109.771,-44.579,178.608,6.057,149.500
C03265=1137.623,-109.521,-44.587,178.610,6.058,149.500
C03266=1137.617,-109.271,-44.597,178.612,6.059,149.499
C03267=1137.611,-109.021,-44.605,178.614,6.059,149.499
C03268=1137.606,-108.771,-44.614,178.616,6.059,149.498
C03269=1137.601,-108.521,-44.623,178.617,6.059,149.498
C03270=1137.596,-108.271,-44.632,178.620,6.060,149.497
C03271=1137.590,-108.022,-44.640,178.621,6.060,149.497
C03272=1137.585,-107.772,-44.649,178.623,6.061,149.496
C03273=1137.580,-107.523,-44.658,178.626,6.062,149.496
C03274=1137.575,-107.273,-44.667,178.627,6.062,149.495
C03275=1137.569,-107.023,-44.676,178.629,6.062,149.495
C03276=1137.564,-106.774,-44.684,178.632,6.063,149.494
C03277=1137.558,-106.524,-44.693,178.634,6.063,149.494
C03278=1137.553,-106.274,-44.703,178.636,6.063,149.493
C03279=1137.547,-106.024,-44.711,178.638,6.063,149.493
C03280=1137.542,-105.774,-44.720,178.640,6.064,149.492
C03281=1137.537,-105.524,-44.729,178.642,6.065,149.492
C03282=1137.531,-105.275,-44.738,178.644,6.065,149.491
C03283=1137.526,-105.025,-44.747,178.646,6.066,149.491
C03284=1137.521,-104.775,-44.756,178.647,6.065,149.490
C03285=1137.516,-104.526,-44.764,178.650,6.066,149.490
C03286=1137.510,-104.275,-44.774,178.652,6.067,149.489
C03287=1137.505,-104.025,-44.783,178.653,6.067,149.489
C03288=1137.500,-103.776,-44.792,178.656,6.068,149.488
C03289=1137.494,-103.527,-44.800,178.658,6.067,149.487
C03290=1137.488,-103.254,-44.810,178.660,6.068,149.487
C03291=1137.482,-102.981,-44.819,178.662,6.069,149.486
C03292=1137.477,-102.709,-44.830,178.664,6.070,149.486
C03293=1137.471,-102.437,-44.839,178.667,6.070,149.485
C03294=1137.465,-102.187,-44.849,178.668,6.070,149.485
C03295=1137.460,-101.937,-44.857,178.671,6.071,149.484
C03296=1137.454,-101.688,-44.866,178.672,6.071,149.484
C03297=1137.449,-101.438,-44.875,178.674,6.071,149.483
C03298=1137.444,-101.189,-44.884,178.677,6.072,149.483
C03299=1137.439,-100.939,-44.893,178.678,6.072,149.482
C03300=1137.433,-100.689,-44.903,178.680,6.073,149.482
C03301=1137.428,-100.439,-44.912,178.683,6.073,149.481
C03302=1137.423,-100.189,-44.921,178.684,6.073,149.481
C03303=1137.417,-99.939,-44.930,178.687,6.074,149.480
C03304=1137.412,-99.689,-44.939,178.689,6.075,149.480
C03305=1137.406,-99.440,-44.948,178.691,6.075,149.479
C03306=1137.401,-99.191,-44.957,178.693,6.075,149.479
C03307=1137.396,-98.941,-44.966,178.694,6.075,149.478
C03308=1137.390,-98.691,-44.976,178.697,6.076,149.478
C03309=1137.385,-98.441,-44.984,178.699,6.077,149.477
C03310=1137.379,-98.191,-44.993,178.700,6.077,149.477
C03311=1137.374,-97.941,-45.002,178.703,6.077,149.476
C03312=1137.369,-97.691,-45.012,178.705,6.078,149.476
C03313=1137.364,-97.442,-45.021,178.707,6.078,149.475
C03314=1137.358,-97.192,-45.030,178.709,6.079,149.475
C03315=1137.352,-96.942,-45.040,178.711,6.079,149.474
C03316=1137.347,-96.692,-45.049,178.713,6.079,149.474
C03317=1137.342,-96.443,-45.058,178.715,6.080,149.473
C03318=1137.336,-96.193,-45.067,178.717,6.081,149.473
C03319=1137.331,-95.943,-45.076,178.719,6.081,149.472
C03320=1137.326,-95.693,-45.085,178.721,6.081,149.472
C03321=1137.320,-95.444,-45.094,178.724,6.082,149.471
C03322=1137.315,-95.194,-45.104,178.725,6.082,149.471
C03323=1137.310,-94.944,-45.113,178.728,6.083,149.470
C03324=1137.305,-94.694,-45.122,178.730,6.083,149.470
C03325=1137.299,-94.444,-45.132,178.731,6.083,149.469
C03326=1137.294,-94.195,-45.141,178.734,6.084,149.469
C03327=1137.289,-93.945,-45.150,178.736,6.085,149.468
C03328=1137.283,-93.695,-45.160,178.737,6.085,149.468
C03329=1137.278,-93.446,-45.169,178.740,6.085,149.467
C03330=1137.272,-93.195,-45.179,178.742,6.086,149.466
C03331=1137.267,-92.946,-45.188,178.744,6.086,149.466
C03332=1137.262,-92.696,-45.197,178.746,6.087,149.465
C03333=1137.256,-92.446,-45.207,178.748,6.087,149.465
C03334=1137.251,-92.196,-45.216,178.750,6.087,149.464
C03335=1137.246,-91.947,-45.225,178.752,6.088,149.464
C03336=1137.240,-91.697,-45.235,178.755,6.088,149.463
C03337=1137.235,-91.447,-45.244,178.756,6.088,149.463
C03338=1137.229,-91.198,-45.254,178.758,6.089,149.462
C03339=1137.224,-90.948,-45.263,178.761,6.090,149.462
C03340=1137.219,-90.698,-45.272,178.762,6.090,149.461
C03341=1137.213,-90.448,-45.282,178.764,6.091,149.461
C03342=1137.208,-90.198,-45.291,178.767,6.091,149.460
C03343=1137.202,-89.948,-45.300,178.769,6.091,149.460
C03344=1137.197,-89.699,-45.310,178.771,6.092,149.459
C03345=1137.192,-89.449,-45.319,178.773,6.092,149.459
C03346=1137.187,-89.200,-45.329,178.775,6.093,149.458
C03347=1137.182,-88.950,-45.338,178.777,6.093,149.458
C03348=1137.176,-88.700,-45.347,178.779,6.094,149.457
C03349=1137.171,-88.450,-45.357,178.781,6.095,149.457
C03350=1137.165,-88.200,-45.367,178.783,6.094,149.456
C03351=1137.161,-87.950,-45.376,178.786,6.095,149.456
C03352=1137.155,-87.700,-45.386,178.788,6.096,149.455
C03353=1137.150,-87.451,-45.396,178.789,6.096,149.455
C03354=1137.144,-87.201,-45.405,178.792,6.096,149.454
C03355=1137.139,-86.952,-45.415,178.794,6.097,149.454
C03356=1137.133,-86.701,-45.424,178.796,6.098,149.453
C03357=1137.128,-86.452,-45.434,178.798,6.098,149.452
C03358=1137.122,-86.202,-45.443,178.800,6.098,149.452
C03359=1137.118,-85.953,-45.453,178.802,6.099,149.451
C03360=1137.112,-85.703,-45.462,178.804,6.099,149.451
C03361=1137.107,-85.453,-45.472,178.806,6.100,149.450
C03362=1137.101,-85.202,-45.482,178.809,6.100,149.450
C03363=1137.097,-84.953,-45.491,178.811,6.101,149.449
C03364=1137.091,-84.703,-45.501,178.813,6.101,149.449
C03365=1137.086,-84.454,-45.511,178.815,6.102,149.448
C03366=1137.080,-84.204,-45.520,178.817,6.102,149.448
C03367=1137.075,-83.954,-45.530,178.819,6.102,149.447
C03368=1137.069,-83.704,-45.539,178.821,6.103,149.447
C03369=1137.064,-83.455,-45.549,178.823,6.103,149.446
C03370=1137.059,-83.206,-45.559,178.826,6.104,149.446
C03371=1137.054,-82.955,-45.568,178.827,6.104,149.445
C03372=1137.049,-82.705,-45.578,178.829,6.105,149.445
C03373=1137.043,-82.455,-45.588,178.832,6.106,149.444
C03374=1137.038,-82.206,-45.598,178.834,6.106,149.443
C03375=1137.032,-81.957,-45.608,178.836,6.106,149.443
C03376=1137.027,-81.707,-45.617,178.838,6.107,149.443
C03377=1137.021,-81.457,-45.627,178.840,6.108,149.442
C03378=1137.017,-81.207,-45.636,178.842,6.108,149.442
C03379=1137.011,-80.957,-45.646,178.845,6.108,149.441
C03380=1137.006,-80.707,-45.657,178.847,6.109,149.440
C03381=1137.000,-80.458,-45.665,178.849,6.109,149.440
C03382=1136.995,-80.208,-45.676,178.851,6.109,149.439
C03383=1136.989,-79.959,-45.686,178.853,6.110,149.439
C03384=1136.985,-79.708,-45.695,178.855,6.111,149.438
C03385=1136.979,-79.458,-45.705,178.858,6.111,149.438
C03386=1136.974,-79.209,-45.715,178.859,6.111,149.437
C03387=1136.968,-78.959,-45.724,178.861,6.112,149.437
C03388=1136.963,-78.710,-45.735,178.864,6.113,149.436
C03389=1136.958,-78.460,-45.744,178.866,6.114,149.436
C03390=1136.953,-78.209,-45.754,178.868,6.113,149.435
C03391=1136.947,-77.960,-45.764,178.870,6.114,149.435
C03392=1136.942,-77.711,-45.774,178.872,6.115,149.434
C03393=1136.937,-77.461,-45.784,178.874,6.115,149.434
C03394=1136.930,-77.189,-45.795,178.877,6.116,149.433
C03395=1136.925,-76.918,-45.806,178.879,6.116,149.432
C03396=1136.919,-76.646,-45.816,178.881,6.116,149.432
C03397=1136.913,-76.375,-45.827,178.884,6.117,149.431
C03398=1136.907,-76.125,-45.838,178.886,6.118,149.431
C03399=1136.902,-75.875,-45.846,178.888,6.118,149.430
C03400=1136.897,-75.625,-45.857,178.890,6.119,149.430
C03401=1136.892,-75.376,-45.867,178.892,6.119,149.429
C03402=1136.887,-75.126,-45.877,178.894,6.119,149.429
C03403=1136.881,-74.877,-45.887,178.897,6.120,149.428
C03404=1136.875,-74.627,-45.897,178.899,6.121,149.428
C03405=1136.870,-74.376,-45.907,178.900,6.121,149.427
C03406=1136.866,-74.127,-45.917,178.903,6.121,149.426
C03407=1136.860,-73.878,-45.927,178.905,6.122,149.426
C03408=1136.854,-73.628,-45.937,178.907,6.123,149.425
C03409=1136.849,-73.378,-45.948,178.910,6.124,149.425
C03410=1136.844,-73.128,-45.957,178.912,6.123,149.424
C03411=1136.839,-72.878,-45.967,178.914,6.124,149.424
C03412=1136.833,-72.629,-45.977,178.916,6.125,149.423
C03413=1136.828,-72.379,-45.988,178.918,6.125,149.423
C03414=1136.822,-72.129,-45.998,178.920,6.125,149.422
C03415=1136.818,-71.880,-46.007,178.923,6.126,149.422
C03416=1136.813,-71.630,-46.018,178.925,6.127,149.421
C03417=1136.807,-71.380,-46.028,178.927,6.127,149.421
C03418=1136.801,-71.131,-46.038,178.929,6.128,149.420
C03419=1136.796,-70.881,-46.049,178.931,6.128,149.420
C03420=1136.791,-70.630,-46.058,178.933,6.128,149.419
C03421=1136.786,-70.381,-46.068,178.936,6.129,149.419
C03422=1136.780,-70.131,-46.078,178.938,6.130,149.418
C03423=1136.775,-69.881,-46.089,178.940,6.131,149.418
C03424=1136.769,-69.632,-46.099,178.942,6.130,149.417
C03425=1136.764,-69.382,-46.109,178.944,6.131,149.416
C03426=1136.759,-69.132,-46.119,178.946,6.132,149.416
C03427=1136.754,-68.883,-46.129,178.949,6.133,149.415
C03428=1136.748,-68.633,-46.140,178.951,6.133,149.415
C03429=1136.743,-68.383,-46.150,178.953,6.133,149.414
C03430=1136.738,-68.133,-46.160,178.955,6.134,149.414
C03431=1136.732,-67.884,-46.171,178.957,6.135,149.413
C03432=1136.726,-67.634,-46.181,178.959,6.135,149.413
C03433=1136.722,-67.384,-46.191,178.962,6.136,149.412
C03434=1136.717,-67.135,-46.201,178.964,6.136,149.412
C03435=1136.712,-66.884,-46.212,178.966,6.136,149.411
C03436=1136.706,-66.635,-46.222,178.968,6.137,149.411
C03437=1136.700,-66.385,-46.232,178.971,6.138,149.410
C03438=1136.695,-66.135,-46.243,178.973,6.138,149.409
C03439=1136.690,-65.886,-46.253,178.975,6.139,149.409
C03440=1136.684,-65.636,-46.263,178.977,6.139,149.408
C03441=1136.680,-65.386,-46.274,178.979,6.139,149.408
C03442=1136.674,-65.137,-46.285,178.982,6.140,149.407
C03443=1136.668,-64.887,-46.295,178.984,6.141,149.407
C03444=1136.663,-64.637,-46.305,178.986,6.142,149.406
C03445=1136.659,-64.388,-46.315,178.989,6.142,149.406
C03446=1136.654,-64.138,-46.326,178.990,6.142,149.405
C03447=1136.648,-63.888,-46.336,178.992,6.143,149.405
C03448=1136.642,-63.638,-46.346,178.995,6.144,149.404
C03449=1136.637,-63.388,-46.357,178.997,6.144,149.403
C03450=1136.632,-63.139,-46.367,179.000,6.145,149.403
C03451=1136.627,-62.889,-46.378,179.002,6.146,149.403
C03452=1136.621,-62.639,-46.388,179.003,6.145,149.402
C03453=1136.616,-62.390,-46.398,179.006,6.146,149.402
C03454=1136.611,-62.140,-46.409,179.008,6.147,149.401
C03455=1136.605,-61.890,-46.419,179.010,6.147,149.400
C03456=1136.601,-61.641,-46.430,179.013,6.148,149.400
C03457=1136.595,-61.391,-46.441,179.015,6.149,149.399
C03458=1136.590,-61.141,-46.451,179.017,6.149,149.399
C03459=1136.584,-60.891,-46.461,179.019,6.149,149.398
C03460=1136.579,-60.642,-46.472,179.021,6.150,149.398
C03461=1136.574,-60.392,-46.483,179.024,6.150,149.397
C03462=1136.568,-60.143,-46.493,179.026,6.151,149.397
C03463=1136.563,-59.892,-46.504,179.028,6.152,149.396
C03464=1136.558,-59.643,-46.514,179.030,6.153,149.396
C03465=1136.553,-59.393,-46.525,179.033,6.152,149.395
C03466=1136.548,-59.144,-46.535,179.035,6.153,149.394
C03467=1136.543,-58.893,-46.546,179.037,6.154,149.394
C03468=1136.537,-58.644,-46.556,179.039,6.155,149.393
C03469=1136.532,-58.394,-46.568,179.042,6.155,149.393
C03470=1136.526,-58.144,-46.578,179.044,6.156,149.392
C03471=1136.521,-57.894,-46.589,179.046,6.157,149.392
C03472=1136.516,-57.645,-46.600,179.048,6.157,149.391
C03473=1136.511,-57.395,-46.610,179.050,6.157,149.391
C03474=1136.505,-57.145,-46.621,179.053,6.158,149.390
C03475=1136.500,-56.896,-46.632,179.055,6.158,149.390
C03476=1136.495,-56.646,-46.642,179.057,6.159,149.389
C03477=1136.490,-56.396,-46.653,179.060,6.160,149.388
C03478=1136.484,-56.147,-46.664,179.062,6.160,149.388
C03479=1136.479,-55.897,-46.674,179.064,6.161,149.388
C03480=1136.473,-55.647,-46.685,179.066,6.161,149.387
C03481=1136.468,-55.397,-46.696,179.068,6.162,149.386
C03482=1136.463,-55.148,-46.707,179.070,6.162,149.386
C03483=1136.458,-54.898,-46.718,179.073,6.163,149.385
C03484=1136.453,-54.649,-46.728,179.075,6.163,149.385
C03485=1136.448,-54.398,-46.739,179.078,6.164,149.384
C03486=1136.442,-54.149,-46.750,179.080,6.165,149.384
C03487=1136.437,-53.899,-46.760,179.082,6.166,149.383
C03488=1136.431,-53.650,-46.772,179.084,6.165,149.383
C03489=1136.426,-53.400,-46.782,179.086,6.166,149.382
C03490=1136.421,-53.151,-46.793,179.088,6.167,149.382
C03491=1136.416,-52.900,-46.804,179.091,6.167,149.381
C03492=1136.411,-52.650,-46.814,179.093,6.168,149.380
C03493=1136.405,-52.401,-46.826,179.095,6.169,149.380
C03494=1136.400,-52.151,-46.836,179.098,6.170,149.379
C03495=1136.395,-51.902,-46.847,179.100,6.170,149.379
C03496=1136.390,-51.652,-46.858,179.102,6.171,149.378
C03497=1136.384,-51.403,-46.869,179.105,6.172,149.378
C03498=1136.379,-51.132,-46.881,179.107,6.172,149.377
C03499=1136.373,-50.860,-46.893,179.110,6.173,149.377
C03500=1136.367,-50.590,-46.904,179.112,6.173,149.376
C03501=1136.362,-50.319,-46.916,179.114,6.174,149.375
C03502=1136.356,-50.070,-46.928,179.117,6.175,149.375
C03503=1136.351,-49.820,-46.938,179.119,6.175,149.374
C03504=1136.346,-49.570,-46.949,179.121,6.176,149.374
C03505=1136.340,-49.320,-46.960,179.123,6.176,149.373
C03506=1136.335,-49.071,-46.972,179.125,6.177,149.373
C03507=1136.329,-48.821,-46.982,179.128,6.177,149.372
C03508=1136.325,-48.571,-46.993,179.130,6.178,149.372
C03509=1136.319,-48.321,-47.005,179.132,6.178,149.371
C03510=1136.314,-48.072,-47.015,179.135,6.179,149.370
C03511=1136.309,-47.822,-47.026,179.137,6.180,149.370
C03512=1136.303,-47.572,-47.038,179.139,6.180,149.369
C03513=1136.298,-47.323,-47.049,179.141,6.181,149.369
C03514=1136.293,-47.073,-47.060,179.144,6.182,149.368
C03515=1136.287,-46.823,-47.071,179.146,6.182,149.368
C03516=1136.282,-46.574,-47.082,179.149,6.183,149.367
C03517=1136.278,-46.324,-47.093,179.151,6.184,149.367
C03518=1136.271,-46.074,-47.104,179.153,6.184,149.366
C03519=1136.266,-45.825,-47.115,179.155,6.184,149.366
C03520=1136.262,-45.575,-47.127,179.158,6.185,149.365
C03521=1136.255,-45.325,-47.137,179.160,6.185,149.364
C03522=1136.251,-45.075,-47.149,179.162,6.186,149.364
C03523=1136.246,-44.826,-47.160,179.164,6.187,149.364
C03524=1136.240,-44.576,-47.171,179.167,6.187,149.363
C03525=1136.235,-44.326,-47.182,179.169,6.188,149.362
C03526=1136.230,-44.077,-47.193,179.171,6.189,149.362
C03527=1136.224,-43.827,-47.204,179.174,6.189,149.361
C03528=1136.219,-43.577,-47.215,179.176,6.190,149.361
C03529=1136.214,-43.327,-47.227,179.178,6.191,149.360
C03530=1136.209,-43.078,-47.238,179.181,6.191,149.360
C03531=1136.204,-42.828,-47.249,179.183,6.192,149.359
C03532=1136.198,-42.578,-47.261,179.185,6.193,149.359
C03533=1136.193,-42.329,-47.272,179.188,6.194,149.358
C03534=1136.187,-42.079,-47.284,179.190,6.194,149.357
C03535=1136.183,-41.830,-47.295,179.192,6.195,149.357
C03536=1136.178,-41.579,-47.305,179.195,6.196,149.356
C03537=1136.172,-41.330,-47.317,179.197,6.196,149.356
C03538=1136.167,-41.081,-47.328,179.199,6.197,149.355
C03539=1136.162,-40.831,-47.340,179.202,6.197,149.355
C03540=1136.157,-40.581,-47.351,179.204,6.197,149.354
C03541=1136.151,-40.331,-47.362,179.206,6.198,149.354
C03542=1136.146,-40.082,-47.373,179.208,6.199,149.353
C03543=1136.140,-39.832,-47.385,179.210,6.199,149.353
C03544=1136.136,-39.582,-47.397,179.213,6.200,149.352
C03545=1136.130,-39.333,-47.408,179.215,6.201,149.351
C03546=1136.125,-39.083,-47.419,179.217,6.201,149.351
C03547=1136.120,-38.833,-47.431,179.220,6.202,149.350
C03548=1136.115,-38.583,-47.442,179.222,6.203,149.350
C03549=1136.109,-38.334,-47.453,179.224,6.203,149.349
C03550=1136.104,-38.084,-47.465,179.227,6.204,149.349
C03551=1136.098,-37.834,-47.477,179.229,6.205,149.348
C03552=1136.094,-37.585,-47.488,179.231,6.205,149.348
C03553=1136.088,-37.335,-47.499,179.234,6.206,149.347
C03554=1136.083,-37.086,-47.511,179.236,6.206,149.347
C03555=1136.078,-36.836,-47.523,179.238,6.207,149.346
C03556=1136.073,-36.586,-47.534,179.241,6.208,149.346
C03557=1136.068,-36.336,-47.546,179.243,6.208,149.345
C03558=1136.061,-36.087,-47.557,179.245,6.209,149.344
C03559=1136.057,-35.837,-47.569,179.248,6.210,149.344
C03560=1136.051,-35.587,-47.580,179.250,6.210,149.343
C03561=1136.047,-35.338,-47.592,179.252,6.211,149.343
C03562=1136.041,-35.088,-47.604,179.255,6.212,149.342
C03563=1136.036,-34.839,-47.615,179.257,6.212,149.342
C03564=1136.031,-34.589,-47.626,179.260,6.213,149.341
C03565=1136.025,-34.339,-47.638,179.262,6.214,149.341
C03566=1136.020,-34.089,-47.650,179.264,6.214,149.340
C03567=1136.015,-33.839,-47.662,179.267,6.215,149.339
C03568=1136.010,-33.590,-47.673,179.269,6.216,149.339
C03569=1136.004,-33.341,-47.684,179.271,6.216,149.338
C03570=1135.999,-33.091,-47.696,179.274,6.217,149.338
C03571=1135.994,-32.841,-47.708,179.276,6.218,149.337
C03572=1135.989,-32.591,-47.719,179.278,6.218,149.337
C03573=1135.983,-32.341,-47.731,179.281,6.219,149.336
C03574=1135.979,-32.092,-47.743,179.283,6.220,149.336
C03575=1135.973,-31.842,-47.754,179.285,6.221,149.335
C03576=1135.967,-31.593,-47.767,179.288,6.221,149.334
C03577=1135.963,-31.343,-47.778,179.290,6.222,149.334
C03578=1135.957,-31.093,-47.790,179.292,6.223,149.334
C03579=1135.952,-30.844,-47.802,179.295,6.223,149.333
C03580=1135.947,-30.594,-47.813,179.297,6.224,149.332
C03581=1135.942,-30.344,-47.825,179.299,6.225,149.332
C03582=1135.936,-30.094,-47.837,179.302,6.226,149.331
C03583=1135.932,-29.845,-47.849,179.305,6.226,149.331
C03584=1135.926,-29.596,-47.860,179.307,6.227,149.330
C03585=1135.920,-29.346,-47.872,179.309,6.228,149.330
C03586=1135.915,-29.096,-47.884,179.312,6.228,149.329
C03587=1135.910,-28.846,-47.895,179.314,6.229,149.329
C03588=1135.905,-28.597,-47.908,179.316,6.230,149.328
C03589=1135.900,-28.347,-47.920,179.319,6.230,149.327
C03590=1135.895,-28.097,-47.931,179.321,6.231,149.327
C03591=1135.890,-27.847,-47.943,179.323,6.232,149.326
C03592=1135.884,-27.598,-47.955,179.326,6.232,149.326
C03593=1135.879,-27.348,-47.968,179.328,6.233,149.325
C03594=1135.874,-27.099,-47.979,179.330,6.234,149.325
C03595=1135.869,-26.849,-47.991,179.333,6.234,149.324
C03596=1135.864,-26.599,-48.003,179.335,6.235,149.324
C03597=1135.858,-26.349,-48.015,179.337,6.236,149.323
C03598=1135.854,-26.100,-48.026,179.340,6.236,149.322
C03599=1135.848,-25.851,-48.038,179.342,6.237,149.322
C03600=1135.843,-25.601,-48.051,179.345,6.238,149.321
C03601=1135.837,-25.351,-48.062,179.347,6.238,149.321
C03602=1135.832,-25.081,-48.075,179.349,6.240,149.320
C03603=1135.827,-24.811,-48.088,179.352,6.240,149.320
C03604=1135.821,-24.541,-48.101,179.354,6.241,149.319
C03605=1135.815,-24.270,-48.115,179.357,6.241,149.319
C03606=1135.810,-24.021,-48.127,179.359,6.242,149.318
C03607=1135.805,-23.771,-48.138,179.362,6.243,149.317
C03608=1135.799,-23.521,-48.150,179.365,6.244,149.317
C03609=1135.794,-23.272,-48.163,179.367,6.245,149.316
C03610=1135.789,-23.022,-48.175,179.369,6.245,149.316
C03611=1135.784,-22.773,-48.187,179.372,6.246,149.315
C03612=1135.778,-22.523,-48.199,179.374,6.247,149.315
C03613=1135.774,-22.273,-48.211,179.377,6.247,149.314
C03614=1135.768,-22.024,-48.223,179.379,6.248,149.314
C03615=1135.763,-21.774,-48.235,179.381,6.249,149.313
C03616=1135.758,-21.525,-48.248,179.384,6.249,149.312
C03617=1135.752,-21.275,-48.260,179.386,6.250,149.312
C03618=1135.747,-21.025,-48.272,179.388,6.251,149.311
C03619=1135.742,-20.775,-48.284,179.391,6.252,149.311
C03620=1135.736,-20.526,-48.296,179.393,6.253,149.310
C03621=1135.731,-20.276,-48.309,179.396,6.254,149.310
C03622=1135.726,-20.026,-48.320,179.398,6.254,149.309
C03623=1135.721,-19.777,-48.333,179.400,6.255,149.309
C03624=1135.715,-19.527,-48.345,179.403,6.256,149.308
C03625=1135.711,-19.278,-48.357,179.405,6.256,149.307
C03626=1135.706,-19.028,-48.369,179.407,6.257,149.307
C03627=1135.700,-18.779,-48.381,179.410,6.258,149.307
